// TIA Portal V15.1 export
// export: Created 2024-06-21T08:41:19.7465003Z, ExportSetting WithDefaults, DisplayName Totally Integrated Automation Portal, DisplayVersion V15.1 Update 5, DisplayName TIA Portal Openness, DisplayVersion V15.1 Update 5, DisplayName SINAMICS Startdrive Advanced, DisplayVersion V15.1, DisplayName G130, G150, S120, S150, SINAMICS MV, S210, DisplayVersion V15.1, DisplayName G110M, G120, G120C, G120D, G120P, DisplayVersion V15.1, DisplayName STEP 7 Professional, DisplayVersion V15.1 Update 5, DisplayName STEP 7 Safety, DisplayVersion V15.1, DisplayName WinCC Professional, DisplayVersion V15.1 Update 5, DisplayName SIMATIC Visualization Architect, DisplayVersion V15.1
FUNCTION_BLOCK "LGBTurnTable2W2S-MoviFitFCPN"   // FB6698, FBD
TITLE = LGBMovUnit2Pos2W2S-MoviFitFCPN / LGBTurnTable2W2S-MoviFitFCPN
{ S7_Optimized_Access := 'TRUE' }
AUTHOR : VCC
FAMILY : Tooling
VERSION : 0.1
// ============================================================================
// This module will be used for a unit with 2 stop positions, 2 speeds and controlled by a 
// SEW MOVIFIT-FC fieldbus frequency converter.
// It will get commands from higher level, evaluate the status of the interlock 
// and give a finished in return when the task is completed.
// It will get commands from higher level, evaluate the status of the interlock 
// and give a finished in return when the task is completed.
// ===========================================================================
// stored: AutoNumber false, IsIECCheckEnabled false, IsRetainMemResEnabled false, MemoryReserve 100, SetENOAutomatically False, UDAEnableTagReadback false
   VAR_INPUT
      I_PosSet { ExternalAccessible := 'False'; ExternalVisible := 'False'; ExternalWritable := 'False'} : Bool;   // Position Set Detection
      I_LowSpeedSet { ExternalAccessible := 'False'; ExternalVisible := 'False'; ExternalWritable := 'False'} : Bool;   // Low Speed Detection Set
      I_PosRes { ExternalAccessible := 'False'; ExternalVisible := 'False'; ExternalWritable := 'False'} : Bool;   // Position Reset Detection
      I_LowSpeedRes { ExternalAccessible := 'False'; ExternalVisible := 'False'; ExternalWritable := 'False'} : Bool;   // Low Speed Detection Reset
      I_SetBegin { ExternalAccessible := 'False'; ExternalVisible := 'False'; ExternalWritable := 'False'} : Bool;   // Function Set begin selection
      I_ResBegin { ExternalAccessible := 'False'; ExternalVisible := 'False'; ExternalWritable := 'False'} : Bool;   // Function Reset begin selection
      I_PBSet { ExternalAccessible := 'False'; ExternalVisible := 'False'; ExternalWritable := 'False'} : Bool;   // Push button for Set direction used in manual
      I_PBReset { ExternalAccessible := 'False'; ExternalVisible := 'False'; ExternalWritable := 'False'} : Bool;   // Push button for reset direcion used in manual
      I_SetIntlkOK { ExternalAccessible := 'False'; ExternalVisible := 'False'; ExternalWritable := 'False'} : Bool;   // Set Interlock
      I_ResIntlkOK { ExternalAccessible := 'False'; ExternalVisible := 'False'; ExternalWritable := 'False'} : Bool;   // Reset Interlock
      I_MotorProtection { ExternalAccessible := 'False'; ExternalVisible := 'False'; ExternalWritable := 'False'} : Bool;   // Motor protection
      I_ReleaseBrake { ExternalAccessible := 'False'; ExternalVisible := 'False'; ExternalWritable := 'False'} : Bool;   // Release brake
      I_SafetyOk { ExternalAccessible := 'False'; ExternalVisible := 'False'; ExternalWritable := 'False'} : Bool;   // Safety Ok
      I_MotionStopOk { ExternalAccessible := 'False'; ExternalVisible := 'False'; ExternalWritable := 'False'} : Bool;   // Safety Ok / The motion stop is Ok
      I_LowSpeed { ExternalAccessible := 'False'; ExternalVisible := 'False'; ExternalWritable := 'False'} : Real;   // Low speed Value (set-up %)
      I_HighSpeed { ExternalAccessible := 'False'; ExternalVisible := 'False'; ExternalWritable := 'False'} : Real;   // High speed Value (set-up %)
      I_SafetyStatusWord { ExternalAccessible := 'False'; ExternalVisible := 'False'; ExternalWritable := 'False'} : Word;   // Safety Status
      I_SafetyControlWord { ExternalAccessible := 'False'; ExternalVisible := 'False'; ExternalWritable := 'False'} : Word;   // Safety Control Word
   END_VAR
   VAR_OUTPUT
      O_SumPosSet { ExternalAccessible := 'False'; ExternalVisible := 'False'; ExternalWritable := 'False'} : Bool;   // Summary In Position Set
      O_SumPosRes { ExternalAccessible := 'False'; ExternalVisible := 'False'; ExternalWritable := 'False'} : Bool;   // Summary In Position Reset
      O_ReleaseBrake { ExternalAccessible := 'False'; ExternalVisible := 'False'; ExternalWritable := 'False'} : Bool;   // Release the brake of the motor
      O_Active { ExternalAccessible := 'False'; ExternalVisible := 'False'; ExternalWritable := 'False'} : Bool;   // Motor Active
      O_FuncRunning { ExternalAccessible := 'False'; ExternalVisible := 'False'; ExternalWritable := 'False'} : Bool;   // Signal that the function is busy
      O_SetFinished { ExternalAccessible := 'False'; ExternalVisible := 'False'; ExternalWritable := 'False'} : Bool;   // Function Set finished to Master Sequencing
      O_ResFinished { ExternalAccessible := 'False'; ExternalVisible := 'False'; ExternalWritable := 'False'} : Bool;   // Function Reset finished to Master Sequencing
      O_LEDSet { ExternalAccessible := 'False'; ExternalVisible := 'False'; ExternalWritable := 'False'} : Bool;   // Ledindication / Led indication for Set
      O_LEDRes { ExternalAccessible := 'False'; ExternalVisible := 'False'; ExternalWritable := 'False'} : Bool;   // Ledindication / Led indication for Reset
      O_ReadyForOperation { ExternalAccessible := 'False'; ExternalVisible := 'False'; ExternalWritable := 'False'} : Bool;   // Ready for operation
      O_AlarmABCondition { ExternalAccessible := 'False'; ExternalVisible := 'False'; ExternalWritable := 'False'} : Bool;   // Alarm AB Condition
      O_AlarmA { ExternalAccessible := 'False'; ExternalVisible := 'False'; ExternalWritable := 'False'} : Bool;   // Alarm A
      O_AlarmB { ExternalAccessible := 'False'; ExternalVisible := 'False'; ExternalWritable := 'False'} : Bool;   // Alarm B
      O_AlarmC { ExternalAccessible := 'False'; ExternalVisible := 'False'; ExternalWritable := 'False'} : Bool;   // Alarm C
      O_AlarmD { ExternalAccessible := 'False'; ExternalVisible := 'False'; ExternalWritable := 'False'} : Bool;   // Alarm D
      H_AlarmDWord { ExternalAccessible := 'False'; ExternalVisible := 'False'; ExternalWritable := 'False'} : DWord;   // Alarm Word
   END_VAR
   VAR_IN_OUT
      IO_Modes : "Modes";   // Modes
      H_HMI : "H_HMI";   // Animation
      "H_GBMovUnit2Pos2W2S-MoviFitFCPN" : "H_GBTurnTable2W2S-MoviFitFCPN";   // Animation
      C_Config : "TurnTable2W2S-MoviFitFCPNConfig";   // Config
   END_VAR
   VAR
      _MovFunc2Pos2s { ExternalAccessible := 'False'; ExternalVisible := 'False'; ExternalWritable := 'False'} : "LMovFnc2Pos2S";   // FB
      _StopPos { ExternalAccessible := 'False'; ExternalVisible := 'False'; ExternalWritable := 'False'} : "L2StopPos";   // FB
      _Motor { ExternalAccessible := 'False'; ExternalVisible := 'False'; ExternalWritable := 'False'} : "LGBMotor2W2S-MoviFitFCPN";   // FB
      H_FncSelInHMI { ExternalAccessible := 'False'; ExternalVisible := 'False'; ExternalWritable := 'False'} : Bool;
      AA_MotorProtection { ExternalAccessible := 'False'; ExternalVisible := 'False'; ExternalWritable := 'False'} : Bool;   // Motorprotection Not Ok
      AA_SafetySwitch { ExternalAccessible := 'False'; ExternalVisible := 'False'; ExternalWritable := 'False'} : Bool;   // Safety Switch Not Ok
      AB_STO { ExternalAccessible := 'False'; ExternalVisible := 'False'; ExternalWritable := 'False'} : Bool;   // Safety Switch Not Ok / Safety output to drive is active but no response from drive that the safety is ok
      AB_Alarm { ExternalAccessible := 'False'; ExternalVisible := 'False'; ExternalWritable := 'False'} : Bool;   // Frequency Control / Alarm Frequency Control
      AB_LSpeedDetSetMissing { ExternalAccessible := 'False'; ExternalVisible := 'False'; ExternalWritable := 'False'} : Bool;   // Low Speed Detector Set / Low Speed Detection Set Is Missing
      AB_LSpeedDetResMissing { ExternalAccessible := 'False'; ExternalVisible := 'False'; ExternalWritable := 'False'} : Bool;   // Low Speed Detector Reset / Low Speed Detection Reset Is Missing
      AB_KeepPosSetAlm { ExternalAccessible := 'False'; ExternalVisible := 'False'; ExternalWritable := 'False'} : Bool;   // Position Supervision Set Position / Lost Set Position
      AB_KeepPosResAlm { ExternalAccessible := 'False'; ExternalVisible := 'False'; ExternalWritable := 'False'} : Bool;   // Position Supervision Reset Position / Lost Reset Position
      AB_OvtSetAlm { ExternalAccessible := 'False'; ExternalVisible := 'False'; ExternalWritable := 'False'} : Bool;   // Timeout Set / TimeOut Set Direction
      AB_OvtResAlm { ExternalAccessible := 'False'; ExternalVisible := 'False'; ExternalWritable := 'False'} : Bool;   // Timeout Reset / TimeOut Reset Direction
      AB_TwoDetAlm { ExternalAccessible := 'False'; ExternalVisible := 'False'; ExternalWritable := 'False'} : Bool;   // Set Reset Activated Simultaneously / Detection Set & Reset Activated Simultaneously
      AC_KeepPosSetAlm { ExternalAccessible := 'False'; ExternalVisible := 'False'; ExternalWritable := 'False'} : Bool;   // Lost Set Position
      AC_KeepPosResAlm { ExternalAccessible := 'False'; ExternalVisible := 'False'; ExternalWritable := 'False'} : Bool;   // Lost Reset Position
      AC_OvtSetAlm { ExternalAccessible := 'False'; ExternalVisible := 'False'; ExternalWritable := 'False'} : Bool;   // Timeout Set / TimeOut Set Direction
      AC_OvtResAlm { ExternalAccessible := 'False'; ExternalVisible := 'False'; ExternalWritable := 'False'} : Bool;   // Timeout Reset / TimeOut Reset Direction
      AC_TwoDetAlm { ExternalAccessible := 'False'; ExternalVisible := 'False'; ExternalWritable := 'False'} : Bool;   // Set Reset Activated Simultaneously / Detection Set & Reset Activated Simultaneously
      AD_OvtSetWarn { ExternalAccessible := 'False'; ExternalVisible := 'False'; ExternalWritable := 'False'} : Bool;   // Timeout Set / TimeOut Set Direction
      AD_OvtResWarn { ExternalAccessible := 'False'; ExternalVisible := 'False'; ExternalWritable := 'False'} : Bool;   // Timeout Reset / TimeOut Reset Direction
      AD_IntlkSetAlm { ExternalAccessible := 'False'; ExternalVisible := 'False'; ExternalWritable := 'False'} : Bool;   // Interlock Set
      AD_IntlkResAlm { ExternalAccessible := 'False'; ExternalVisible := 'False'; ExternalWritable := 'False'} : Bool;   // Interlock Reset
      AD_Warning { ExternalAccessible := 'False'; ExternalVisible := 'False'; ExternalWritable := 'False'} : Bool;   // Frequency Control / Warning Frequency Control
      AA_NoBusControl { ExternalAccessible := 'False'; ExternalVisible := 'False'; ExternalWritable := 'False'} : Bool;   // Bus control inactive / Bus Control Inactive Frequency Control
      AD_MotionStop { ExternalAccessible := 'False'; ExternalVisible := 'False'; ExternalWritable := 'False'} : Bool;   // Motion Stop
      AC_ConfigCalibrationAlm { ExternalAccessible := 'False'; ExternalVisible := 'False'; ExternalWritable := 'False'} : Bool;   // The Config values for Warming/Alarm time must be ALL zero or ALL different from zero
      AD_CalibrationWarn { ExternalAccessible := 'False'; ExternalVisible := 'False'; ExternalWritable := 'False'} : Bool;   // No High speed selected so Calibration is not possible
      AC_ConfigRampAlm { ExternalAccessible := 'False'; ExternalVisible := 'False'; ExternalWritable := 'False'} : Bool;   // The config value for the ramp is not correct, must be zero or the config values for the calculation of the ramp must be ALL zero
      AC_ConfigRampCalcAlm { ExternalAccessible := 'False'; ExternalVisible := 'False'; ExternalWritable := 'False'} : Bool;   // The config values for the calculation of the ramp must be ALL different from zero
      PODataNotEnabled { ExternalAccessible := 'False'; ExternalVisible := 'False'; ExternalWritable := 'False'} : Bool;   // Bus control inactive
      SafetyOk { ExternalAccessible := 'False'; ExternalVisible := 'False'; ExternalWritable := 'False'} : Bool;   // Safety Ok
      AlarmABCondition { ExternalAccessible := 'False'; ExternalVisible := 'False'; ExternalWritable := 'False'} : Bool;   // Alarm AB Condition
   END_VAR
   VAR RETAIN
      LowSpeedDetSetOk { ExternalAccessible := 'False'; ExternalVisible := 'False'; ExternalWritable := 'False'} : Bool;   // Low speed Set detector ok
      LowSpeedDetResOk { ExternalAccessible := 'False'; ExternalVisible := 'False'; ExternalWritable := 'False'} : Bool;   // Low speed Reset detector ok
   END_VAR
   VAR
      SetPos { ExternalAccessible := 'False'; ExternalVisible := 'False'; ExternalWritable := 'False'} : Bool;   // Set position
      ResPos { ExternalAccessible := 'False'; ExternalVisible := 'False'; ExternalWritable := 'False'} : Bool;   // Reset position
      AlarmA { ExternalAccessible := 'False'; ExternalVisible := 'False'; ExternalWritable := 'False'} : Bool;   // Alarm A
      AlarmB { ExternalAccessible := 'False'; ExternalVisible := 'False'; ExternalWritable := 'False'} : Bool;   // Alarm B
      AlarmC { ExternalAccessible := 'False'; ExternalVisible := 'False'; ExternalWritable := 'False'} : Bool;   // Alarm C
      AlarmD { ExternalAccessible := 'False'; ExternalVisible := 'False'; ExternalWritable := 'False'} : Bool;   // Alarm D
      FuncRunning { ExternalAccessible := 'False'; ExternalVisible := 'False'; ExternalWritable := 'False'} : Bool;   // Function running
      MovFuncAlmCond { ExternalAccessible := 'False'; ExternalVisible := 'False'; ExternalWritable := 'False'} : Bool;   // Move function Alarm Condition
      StopPosAlmCond { ExternalAccessible := 'False'; ExternalVisible := 'False'; ExternalWritable := 'False'} : Bool;   // Stop posistion Alarm Condition
      KeepPosSetAlm { ExternalAccessible := 'False'; ExternalVisible := 'False'; ExternalWritable := 'False'} : Bool;   // Alarm Keep Position Set Position
      KeepPosResAlm { ExternalAccessible := 'False'; ExternalVisible := 'False'; ExternalWritable := 'False'} : Bool;   // Position Supervision Reset Position
      OvtSetAlm { ExternalAccessible := 'False'; ExternalVisible := 'False'; ExternalWritable := 'False'} : Bool;   // Timeout Set
      OvtResAlm { ExternalAccessible := 'False'; ExternalVisible := 'False'; ExternalWritable := 'False'} : Bool;   // Overtime reset Alarm
      TwoDetAlm { ExternalAccessible := 'False'; ExternalVisible := 'False'; ExternalWritable := 'False'} : Bool;   // Set Reset Activated Simultaneously
      OutOfUse { ExternalAccessible := 'False'; ExternalVisible := 'False'; ExternalWritable := 'False'} : Bool;   // Out of use
      MotorLoopAlarmCond { ExternalAccessible := 'False'; ExternalVisible := 'False'; ExternalWritable := 'False'} : Bool;   // Motor loop Alarm Condition
      SafetySwNc { ExternalAccessible := 'False'; ExternalVisible := 'False'; ExternalWritable := 'False'} : Bool;   // Safety switch NC
      InitDirection { ExternalAccessible := 'False'; ExternalVisible := 'False'; ExternalWritable := 'False'} : Bool;   // Init Direction
      ReadyForOperation { ExternalAccessible := 'False'; ExternalVisible := 'False'; ExternalWritable := 'False'} : Bool;   // Motor Loop Ready for operation
      MotorLoopActive { ExternalAccessible := 'False'; ExternalVisible := 'False'; ExternalWritable := 'False'} : Bool;   // Motor Loop Active
      ReleaseBrake { ExternalAccessible := 'False'; ExternalVisible := 'False'; ExternalWritable := 'False'} : Bool;   // Release brake
      CmdSet { ExternalAccessible := 'False'; ExternalVisible := 'False'; ExternalWritable := 'False'} : Bool;   // Command set
      CmdRes { ExternalAccessible := 'False'; ExternalVisible := 'False'; ExternalWritable := 'False'} : Bool;   // DCommand Reset
      MotorCmdHSpdSet { ExternalAccessible := 'False'; ExternalVisible := 'False'; ExternalWritable := 'False'} : Bool;   // Command high speed to motorloop set
      MotorCmdLSpdSet { ExternalAccessible := 'False'; ExternalVisible := 'False'; ExternalWritable := 'False'} : Bool;   // Command low speed to motorloop set
      MotorCmdHSpdRes { ExternalAccessible := 'False'; ExternalVisible := 'False'; ExternalWritable := 'False'} : Bool;   // Command high speed to motorloop reset
      MotorCmdLSpdRes { ExternalAccessible := 'False'; ExternalVisible := 'False'; ExternalWritable := 'False'} : Bool;   // Command low speed to motorloop reset
      DetStopHSpdSetMem { ExternalAccessible := 'False'; ExternalVisible := 'False'; ExternalWritable := 'False'} : Bool;   // Memorisation stop high speed set
      DetStopHSpdResMem { ExternalAccessible := 'False'; ExternalVisible := 'False'; ExternalWritable := 'False'} : Bool;   // Memorisation stop high speed reset
      ManLowSpdSel { ExternalAccessible := 'False'; ExternalVisible := 'False'; ExternalWritable := 'False'} : Bool;   // Low speed Selected in manual
      LowSpeedSetDetMissingCond { ExternalAccessible := 'False'; ExternalVisible := 'False'; ExternalWritable := 'False'} : Bool;   // Low speed detector missing condition set
      LowSpeedResDetMissingCond { ExternalAccessible := 'False'; ExternalVisible := 'False'; ExternalWritable := 'False'} : Bool;   // Low speed detector missing condition reset
      SetIntlkOK { ExternalAccessible := 'False'; ExternalVisible := 'False'; ExternalWritable := 'False'} : Bool;   // Set Interlock
      ResIntlkOK { ExternalAccessible := 'False'; ExternalVisible := 'False'; ExternalWritable := 'False'} : Bool;   // Reset Interlock
      Edge { ExternalAccessible := 'False'; ExternalVisible := 'False'; ExternalWritable := 'False'} : Array[1..8] of Bool;
   END_VAR
   VAR_TEMP
      H_HMITemp : "H_HMI";   // Animation
      HMICMD : "ConvHMICMD";
      H_HMIMotor : "H_HMI";
      TempDInt : DInt;   // Temp DInt
   END_VAR
   VAR_TEMP   // added for the SCL form of the ladder/FBD networks
      _w1 : Bool;
   END_VAR
BEGIN

REGION Network 1: **** 1 - Inputs **** HMI Commands
   // HMI Commands
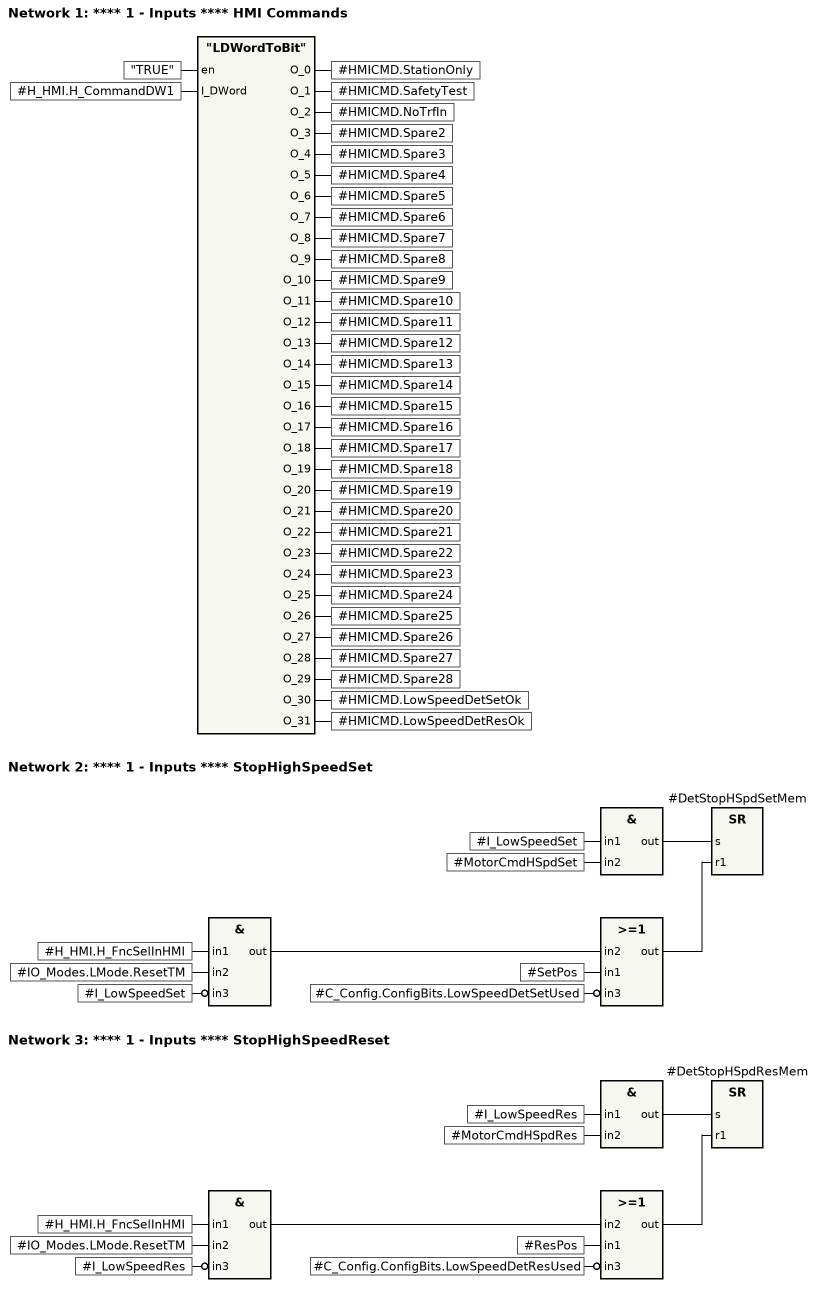
   IF "TRUE" THEN
       "LDWordToBit"(I_DWord := #H_HMI.H_CommandDW1,
                     O_0 => #HMICMD.StationOnly,
                     O_1 => #HMICMD.SafetyTest,
                     O_2 => #HMICMD.NoTrfIn,
                     O_3 => #HMICMD.Spare2,
                     O_4 => #HMICMD.Spare3,
                     O_5 => #HMICMD.Spare4,
                     O_6 => #HMICMD.Spare5,
                     O_7 => #HMICMD.Spare6,
                     O_8 => #HMICMD.Spare7,
                     O_9 => #HMICMD.Spare8,
                     O_10 => #HMICMD.Spare9,
                     O_11 => #HMICMD.Spare10,
                     O_12 => #HMICMD.Spare11,
                     O_13 => #HMICMD.Spare12,
                     O_14 => #HMICMD.Spare13,
                     O_15 => #HMICMD.Spare14,
                     O_16 => #HMICMD.Spare15,
                     O_17 => #HMICMD.Spare16,
                     O_18 => #HMICMD.Spare17,
                     O_19 => #HMICMD.Spare18,
                     O_20 => #HMICMD.Spare19,
                     O_21 => #HMICMD.Spare20,
                     O_22 => #HMICMD.Spare21,
                     O_23 => #HMICMD.Spare22,
                     O_24 => #HMICMD.Spare23,
                     O_25 => #HMICMD.Spare24,
                     O_26 => #HMICMD.Spare25,
                     O_27 => #HMICMD.Spare26,
                     O_28 => #HMICMD.Spare27,
                     O_29 => #HMICMD.Spare28,
                     O_30 => #HMICMD.LowSpeedDetSetOk,
                     O_31 => #HMICMD.LowSpeedDetResOk);
   END_IF;
END_REGION

REGION Network 2: **** 1 - Inputs **** StopHighSpeedSet
   // Stop high speed set memorisation (go to low speed)
   IF #I_LowSpeedSet AND #MotorCmdHSpdSet THEN
       #DetStopHSpdSetMem := TRUE;   // SR flip-flop
   END_IF;
   IF (#H_HMI.H_FncSelInHMI AND #IO_Modes.LMode.ResetTM AND NOT #I_LowSpeedSet) OR #SetPos OR NOT #C_Config.ConfigBits.LowSpeedDetSetUsed THEN
       #DetStopHSpdSetMem := FALSE;
   END_IF;
END_REGION

REGION Network 3: **** 1 - Inputs **** StopHighSpeedReset
   // Stop high speed reset memorisation (go to low speed)
   IF #I_LowSpeedRes AND #MotorCmdHSpdRes THEN
       #DetStopHSpdResMem := TRUE;   // SR flip-flop
   END_IF;
   IF (#H_HMI.H_FncSelInHMI AND #IO_Modes.LMode.ResetTM AND NOT #I_LowSpeedRes) OR #ResPos OR NOT #C_Config.ConfigBits.LowSpeedDetResUsed THEN
       #DetStopHSpdResMem := FALSE;
   END_IF;
END_REGION

REGION Network 4: **** 1 - Inputs **** LowSpeedSet
   // Low speed set detector been on
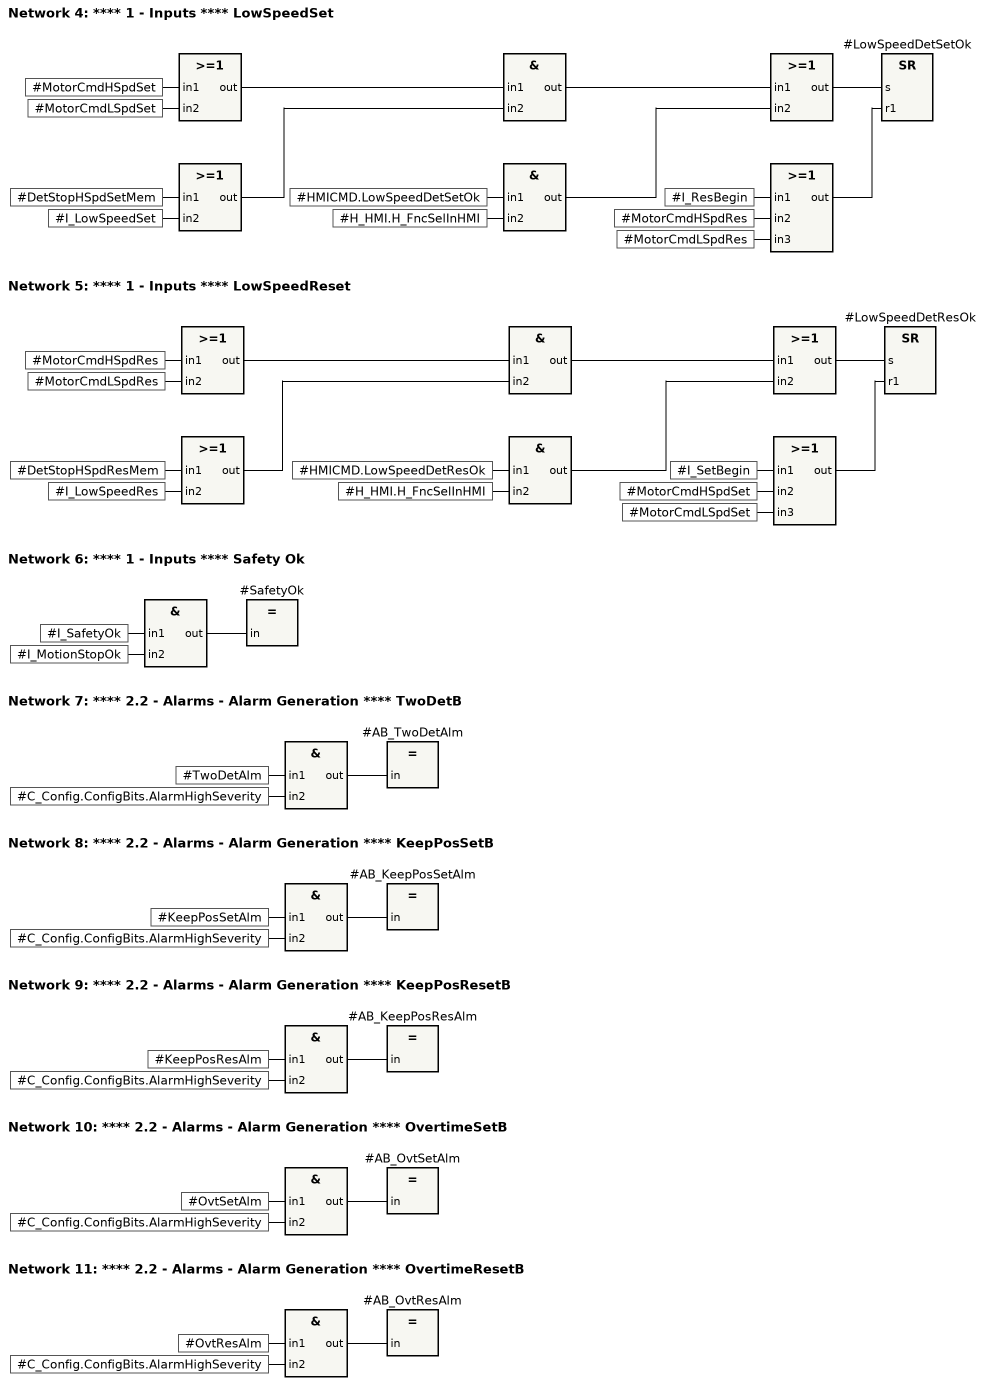
   IF ((#MotorCmdHSpdSet OR #MotorCmdLSpdSet) AND (#DetStopHSpdSetMem OR #I_LowSpeedSet)) OR (#HMICMD.LowSpeedDetSetOk AND #H_HMI.H_FncSelInHMI) THEN
       #LowSpeedDetSetOk := TRUE;   // SR flip-flop
   END_IF;
   IF #I_ResBegin OR #MotorCmdHSpdRes OR #MotorCmdLSpdRes THEN #LowSpeedDetSetOk := FALSE; END_IF;
END_REGION

REGION Network 5: **** 1 - Inputs **** LowSpeedReset
   // Low speed reset detector been on
   IF ((#MotorCmdHSpdRes OR #MotorCmdLSpdRes) AND (#DetStopHSpdResMem OR #I_LowSpeedRes)) OR (#HMICMD.LowSpeedDetResOk AND #H_HMI.H_FncSelInHMI) THEN
       #LowSpeedDetResOk := TRUE;   // SR flip-flop
   END_IF;
   IF #I_SetBegin OR #MotorCmdHSpdSet OR #MotorCmdLSpdSet THEN #LowSpeedDetResOk := FALSE; END_IF;
END_REGION

REGION Network 6: **** 1 - Inputs **** Safety Ok
   #SafetyOk := #I_SafetyOk AND #I_MotionStopOk;
END_REGION

REGION Network 7: **** 2.2 - Alarms - Alarm Generation **** TwoDetB
   // Two Detection B Alarm
   #AB_TwoDetAlm := #TwoDetAlm AND #C_Config.ConfigBits.AlarmHighSeverity;
END_REGION

REGION Network 8: **** 2.2 - Alarms - Alarm Generation **** KeepPosSetB
   // Keep position Set B Alarm
   #AB_KeepPosSetAlm := #KeepPosSetAlm AND #C_Config.ConfigBits.AlarmHighSeverity;
END_REGION

REGION Network 9: **** 2.2 - Alarms - Alarm Generation **** KeepPosResetB
   // Keep position reset B Alarm
   #AB_KeepPosResAlm := #KeepPosResAlm AND #C_Config.ConfigBits.AlarmHighSeverity;
END_REGION

REGION Network 10: **** 2.2 - Alarms - Alarm Generation **** OvertimeSetB
   // Overtime set B Alarm
   #AB_OvtSetAlm := #OvtSetAlm AND #C_Config.ConfigBits.AlarmHighSeverity;
END_REGION

REGION Network 11: **** 2.2 - Alarms - Alarm Generation **** OvertimeResetB
   // Overtime reset B Alarm
   #AB_OvtResAlm := #OvtResAlm AND #C_Config.ConfigBits.AlarmHighSeverity;
END_REGION

REGION Network 12: **** 2.2 - Alarms - Alarm Generation **** TwoDetC
   // Two Detection C Alarm
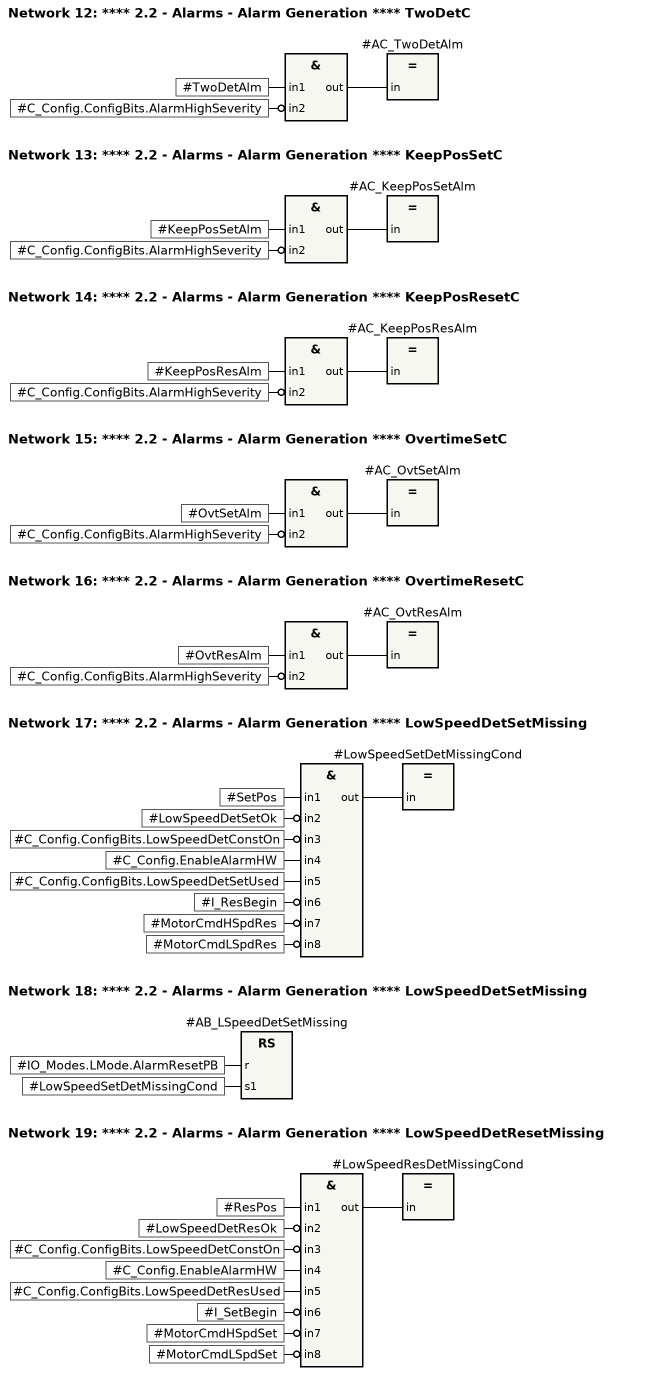
   #AC_TwoDetAlm := #TwoDetAlm AND NOT #C_Config.ConfigBits.AlarmHighSeverity;
END_REGION

REGION Network 13: **** 2.2 - Alarms - Alarm Generation **** KeepPosSetC
   // Keep position Set C Alarm
   #AC_KeepPosSetAlm := #KeepPosSetAlm AND NOT #C_Config.ConfigBits.AlarmHighSeverity;
END_REGION

REGION Network 14: **** 2.2 - Alarms - Alarm Generation **** KeepPosResetC
   // Keep position reset C Alarm
   #AC_KeepPosResAlm := #KeepPosResAlm AND NOT #C_Config.ConfigBits.AlarmHighSeverity;
END_REGION

REGION Network 15: **** 2.2 - Alarms - Alarm Generation **** OvertimeSetC
   // Overtime set C Alarm
   #AC_OvtSetAlm := #OvtSetAlm AND NOT #C_Config.ConfigBits.AlarmHighSeverity;
END_REGION

REGION Network 16: **** 2.2 - Alarms - Alarm Generation **** OvertimeResetC
   // Overtime reset C Alarm
   #AC_OvtResAlm := #OvtResAlm AND NOT #C_Config.ConfigBits.AlarmHighSeverity;
END_REGION

REGION Network 17: **** 2.2 - Alarms - Alarm Generation **** LowSpeedDetSetMissing
   // Alarm LowSpeed detector set missing
   #LowSpeedSetDetMissingCond := #SetPos AND NOT #LowSpeedDetSetOk AND NOT #C_Config.ConfigBits.LowSpeedDetConstOn AND #C_Config.EnableAlarmHW AND #C_Config.ConfigBits.LowSpeedDetSetUsed AND NOT #I_ResBegin AND NOT #MotorCmdHSpdRes AND NOT #MotorCmdLSpdRes;
END_REGION

REGION Network 18: **** 2.2 - Alarms - Alarm Generation **** LowSpeedDetSetMissing
   // Alarm LowSpeed detector set missing
   IF #IO_Modes.LMode.AlarmResetPB THEN
       #AB_LSpeedDetSetMissing := FALSE;   // RS flip-flop
   END_IF;
   IF #LowSpeedSetDetMissingCond THEN #AB_LSpeedDetSetMissing := TRUE; END_IF;
END_REGION

REGION Network 19: **** 2.2 - Alarms - Alarm Generation **** LowSpeedDetResetMissing
   // Alarm LowSpeed detector reset missing
   #LowSpeedResDetMissingCond := #ResPos AND NOT #LowSpeedDetResOk AND NOT #C_Config.ConfigBits.LowSpeedDetConstOn AND #C_Config.EnableAlarmHW AND #C_Config.ConfigBits.LowSpeedDetResUsed AND NOT #I_SetBegin AND NOT #MotorCmdHSpdSet AND NOT #MotorCmdLSpdSet;
END_REGION

REGION Network 20: **** 2.2 - Alarms - Alarm Generation **** LowSpeedDetResetMissing
   // Alarm LowSpeed detector reset missing
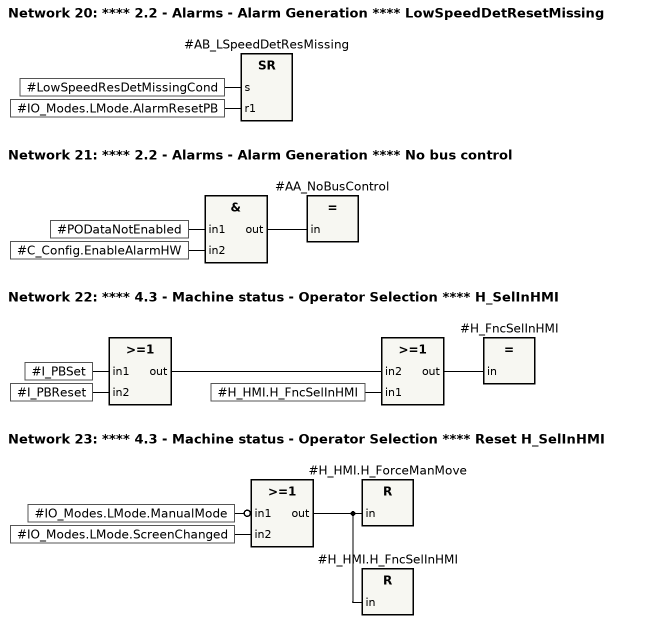
   IF #LowSpeedResDetMissingCond THEN
       #AB_LSpeedDetResMissing := TRUE;   // SR flip-flop
   END_IF;
   IF #IO_Modes.LMode.AlarmResetPB THEN #AB_LSpeedDetResMissing := FALSE; END_IF;
END_REGION

REGION Network 21: **** 2.2 - Alarms - Alarm Generation **** No bus control
   #AA_NoBusControl := #PODataNotEnabled AND #C_Config.EnableAlarmHW;
END_REGION

REGION Network 22: **** 4.3 - Machine status - Operator Selection **** H_SelInHMI
   #H_FncSelInHMI := #I_PBSet OR #I_PBReset OR #H_HMI.H_FncSelInHMI;
END_REGION

REGION Network 23: **** 4.3 - Machine status - Operator Selection **** Reset H_SelInHMI
   // Reset H_SelInHMI
   IF NOT #IO_Modes.LMode.ManualMode OR #IO_Modes.LMode.ScreenChanged THEN
       #H_HMI.H_ForceManMove := FALSE;
       #H_HMI.H_FncSelInHMI := FALSE;
   END_IF;
END_REGION

REGION Network 24: **** 4.6 - Machine Status - Indication **** SetDetIAnim
   // Icon animation
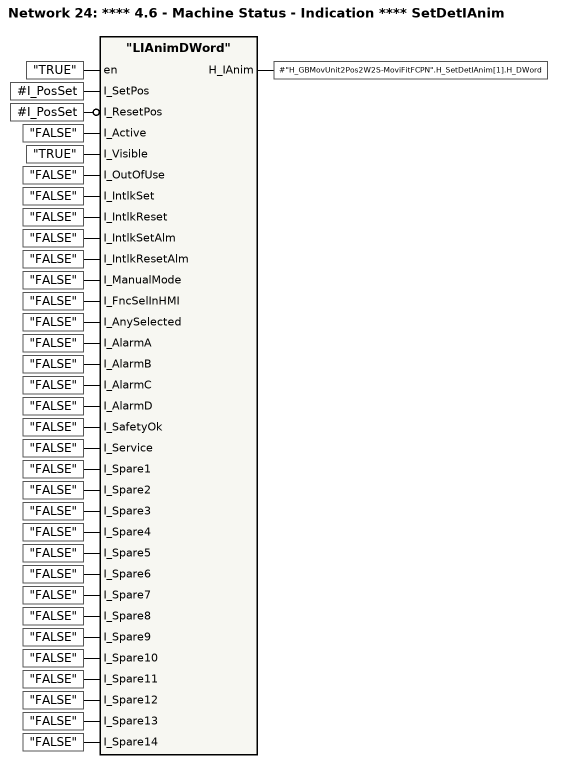
   IF "TRUE" THEN
       "LIAnimDWord"(I_SetPos := #I_PosSet,
                     I_ResetPos := NOT #I_PosSet,
                     I_Active := "FALSE",
                     I_Visible := "TRUE",
                     I_OutOfUse := "FALSE",
                     I_IntlkSet := "FALSE",
                     I_IntlkReset := "FALSE",
                     I_IntlkSetAlm := "FALSE",
                     I_IntlkResetAlm := "FALSE",
                     I_ManualMode := "FALSE",
                     I_FncSelInHMI := "FALSE",
                     I_AnySelected := "FALSE",
                     I_AlarmA := "FALSE",
                     I_AlarmB := "FALSE",
                     I_AlarmC := "FALSE",
                     I_AlarmD := "FALSE",
                     I_SafetyOk := "FALSE",
                     I_Service := "FALSE",
                     I_Spare1 := "FALSE",
                     I_Spare2 := "FALSE",
                     I_Spare3 := "FALSE",
                     I_Spare4 := "FALSE",
                     I_Spare5 := "FALSE",
                     I_Spare6 := "FALSE",
                     I_Spare7 := "FALSE",
                     I_Spare8 := "FALSE",
                     I_Spare9 := "FALSE",
                     I_Spare10 := "FALSE",
                     I_Spare11 := "FALSE",
                     I_Spare12 := "FALSE",
                     I_Spare13 := "FALSE",
                     I_Spare14 := "FALSE",
                     H_IAnim => #"H_GBMovUnit2Pos2W2S-MoviFitFCPN".H_SetDetIAnim[1].H_DWord);
   END_IF;
END_REGION

REGION Network 25: **** 4.6 - Machine Status - Indication **** ResetDetIAnim
   // Icon animation
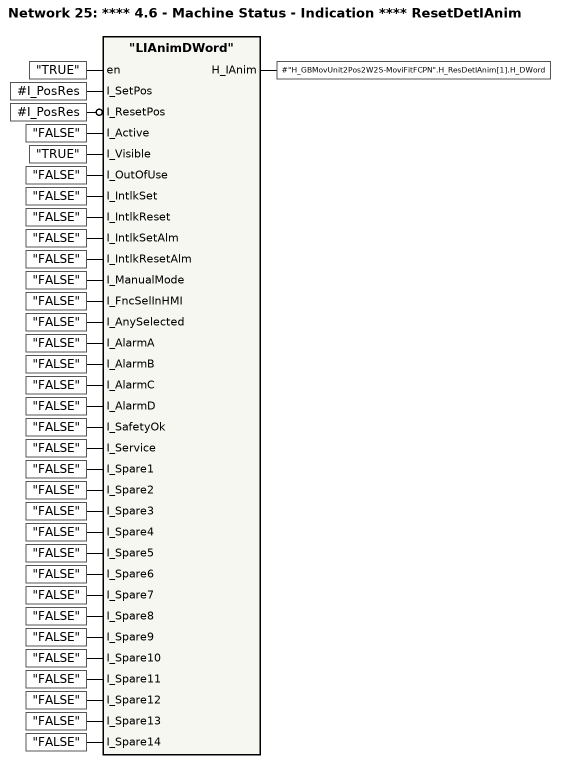
   IF "TRUE" THEN
       "LIAnimDWord"(I_SetPos := #I_PosRes,
                     I_ResetPos := NOT #I_PosRes,
                     I_Active := "FALSE",
                     I_Visible := "TRUE",
                     I_OutOfUse := "FALSE",
                     I_IntlkSet := "FALSE",
                     I_IntlkReset := "FALSE",
                     I_IntlkSetAlm := "FALSE",
                     I_IntlkResetAlm := "FALSE",
                     I_ManualMode := "FALSE",
                     I_FncSelInHMI := "FALSE",
                     I_AnySelected := "FALSE",
                     I_AlarmA := "FALSE",
                     I_AlarmB := "FALSE",
                     I_AlarmC := "FALSE",
                     I_AlarmD := "FALSE",
                     I_SafetyOk := "FALSE",
                     I_Service := "FALSE",
                     I_Spare1 := "FALSE",
                     I_Spare2 := "FALSE",
                     I_Spare3 := "FALSE",
                     I_Spare4 := "FALSE",
                     I_Spare5 := "FALSE",
                     I_Spare6 := "FALSE",
                     I_Spare7 := "FALSE",
                     I_Spare8 := "FALSE",
                     I_Spare9 := "FALSE",
                     I_Spare10 := "FALSE",
                     I_Spare11 := "FALSE",
                     I_Spare12 := "FALSE",
                     I_Spare13 := "FALSE",
                     I_Spare14 := "FALSE",
                     H_IAnim => #"H_GBMovUnit2Pos2W2S-MoviFitFCPN".H_ResDetIAnim[1].H_DWord);
   END_IF;
END_REGION

REGION Network 26: **** 4.6 - Machine Status - Indication **** LSpdDetSetIAnim
   // Icon animation
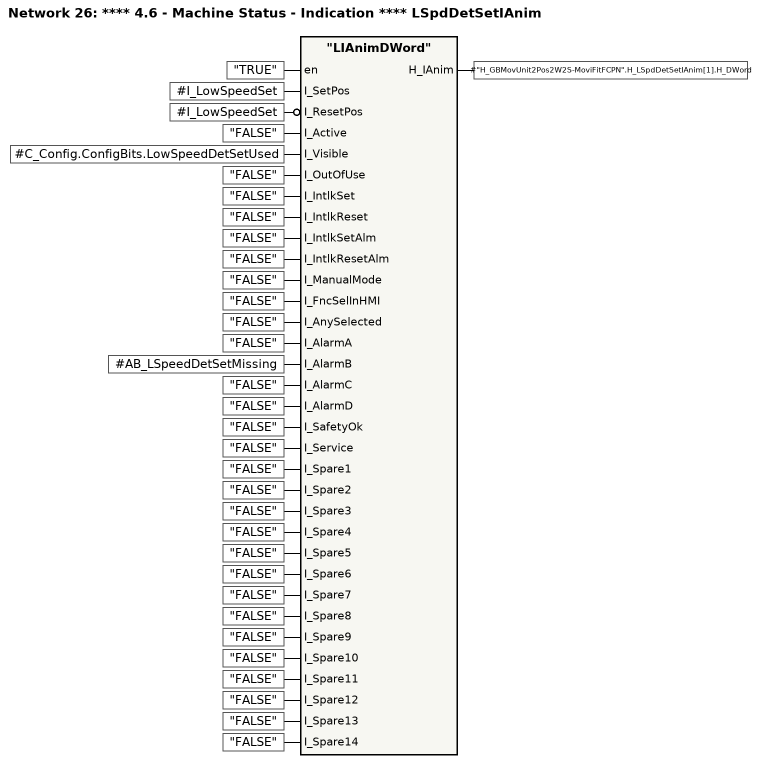
   IF "TRUE" THEN
       "LIAnimDWord"(I_SetPos := #I_LowSpeedSet,
                     I_ResetPos := NOT #I_LowSpeedSet,
                     I_Active := "FALSE",
                     I_Visible := #C_Config.ConfigBits.LowSpeedDetSetUsed,
                     I_OutOfUse := "FALSE",
                     I_IntlkSet := "FALSE",
                     I_IntlkReset := "FALSE",
                     I_IntlkSetAlm := "FALSE",
                     I_IntlkResetAlm := "FALSE",
                     I_ManualMode := "FALSE",
                     I_FncSelInHMI := "FALSE",
                     I_AnySelected := "FALSE",
                     I_AlarmA := "FALSE",
                     I_AlarmB := #AB_LSpeedDetSetMissing,
                     I_AlarmC := "FALSE",
                     I_AlarmD := "FALSE",
                     I_SafetyOk := "FALSE",
                     I_Service := "FALSE",
                     I_Spare1 := "FALSE",
                     I_Spare2 := "FALSE",
                     I_Spare3 := "FALSE",
                     I_Spare4 := "FALSE",
                     I_Spare5 := "FALSE",
                     I_Spare6 := "FALSE",
                     I_Spare7 := "FALSE",
                     I_Spare8 := "FALSE",
                     I_Spare9 := "FALSE",
                     I_Spare10 := "FALSE",
                     I_Spare11 := "FALSE",
                     I_Spare12 := "FALSE",
                     I_Spare13 := "FALSE",
                     I_Spare14 := "FALSE",
                     H_IAnim => #"H_GBMovUnit2Pos2W2S-MoviFitFCPN".H_LSpdDetSetIAnim[1].H_DWord);
   END_IF;
END_REGION

REGION Network 27: **** 4.6 - Machine Status - Indication **** LSpdDetResIAnim
   // Icon animation
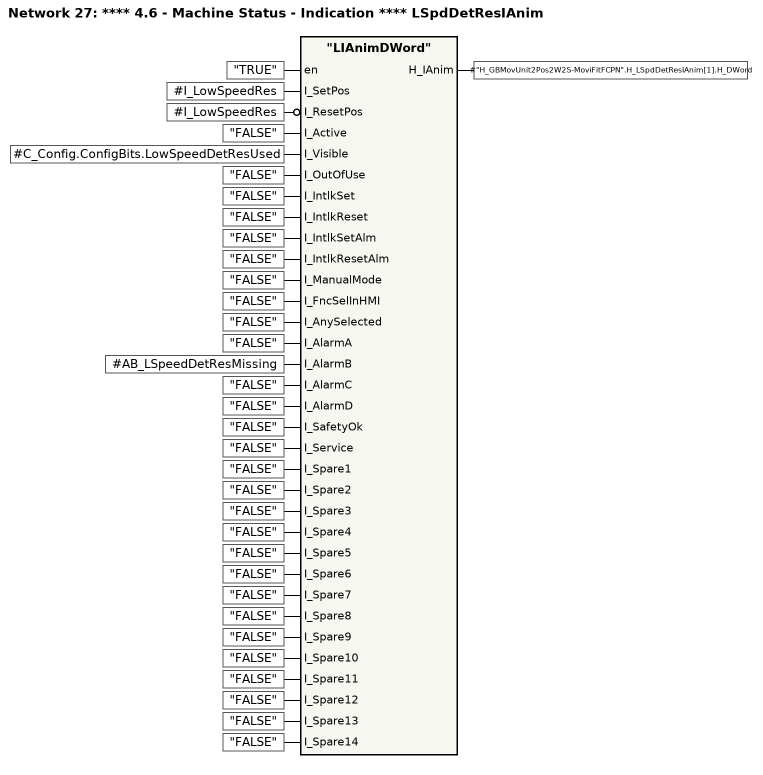
   IF "TRUE" THEN
       "LIAnimDWord"(I_SetPos := #I_LowSpeedRes,
                     I_ResetPos := NOT #I_LowSpeedRes,
                     I_Active := "FALSE",
                     I_Visible := #C_Config.ConfigBits.LowSpeedDetResUsed,
                     I_OutOfUse := "FALSE",
                     I_IntlkSet := "FALSE",
                     I_IntlkReset := "FALSE",
                     I_IntlkSetAlm := "FALSE",
                     I_IntlkResetAlm := "FALSE",
                     I_ManualMode := "FALSE",
                     I_FncSelInHMI := "FALSE",
                     I_AnySelected := "FALSE",
                     I_AlarmA := "FALSE",
                     I_AlarmB := #AB_LSpeedDetResMissing,
                     I_AlarmC := "FALSE",
                     I_AlarmD := "FALSE",
                     I_SafetyOk := "FALSE",
                     I_Service := "FALSE",
                     I_Spare1 := "FALSE",
                     I_Spare2 := "FALSE",
                     I_Spare3 := "FALSE",
                     I_Spare4 := "FALSE",
                     I_Spare5 := "FALSE",
                     I_Spare6 := "FALSE",
                     I_Spare7 := "FALSE",
                     I_Spare8 := "FALSE",
                     I_Spare9 := "FALSE",
                     I_Spare10 := "FALSE",
                     I_Spare11 := "FALSE",
                     I_Spare12 := "FALSE",
                     I_Spare13 := "FALSE",
                     I_Spare14 := "FALSE",
                     H_IAnim => #"H_GBMovUnit2Pos2W2S-MoviFitFCPN".H_LSpdDetResIAnim[1].H_DWord);
   END_IF;
END_REGION

REGION Network 28: **** 4.6 - Machine Status - Indication **** Icon Animation
   // Icon animation
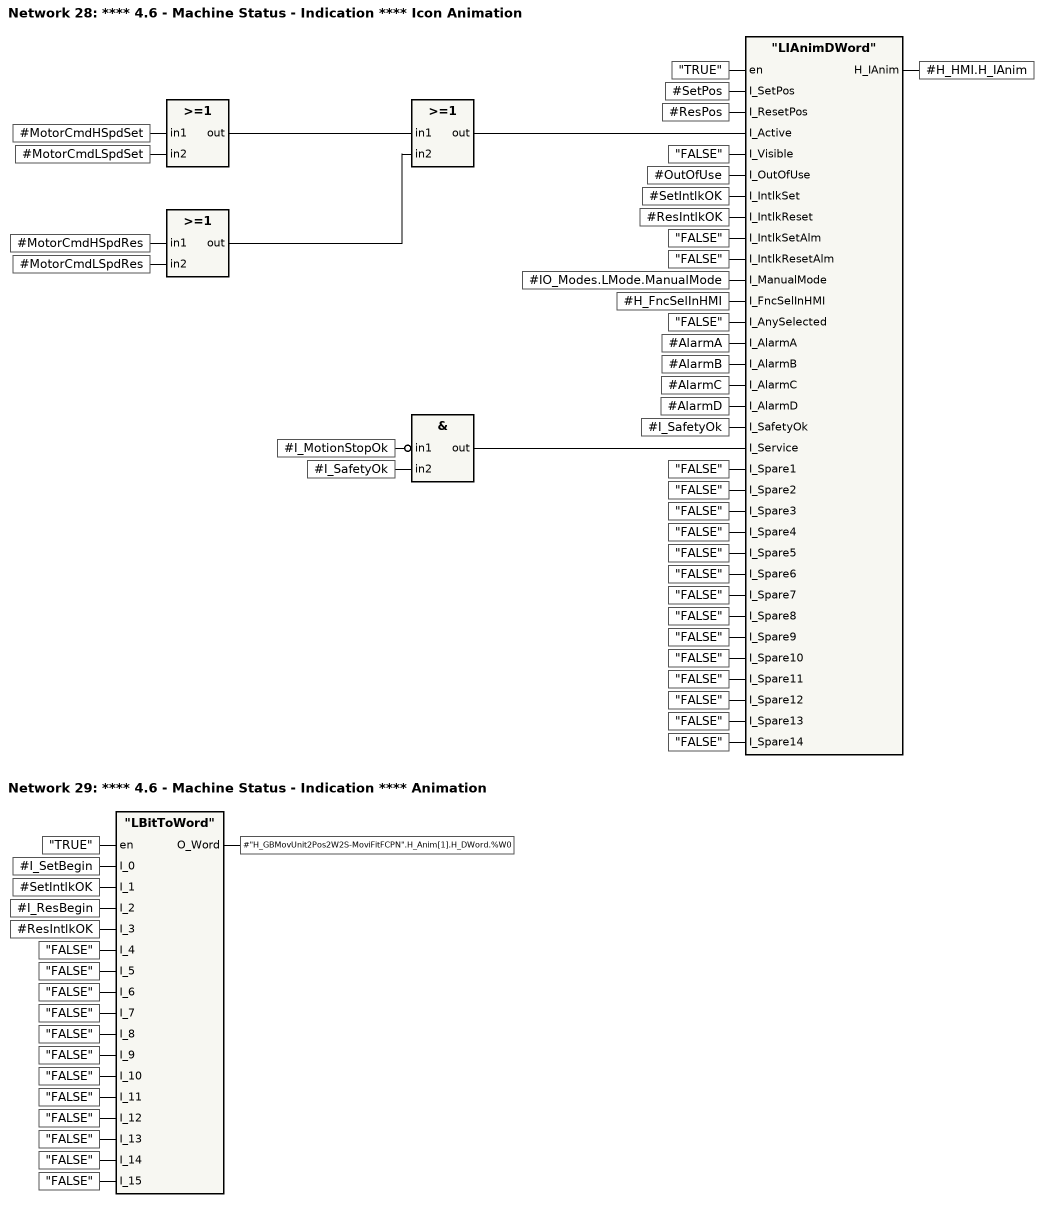
   IF "TRUE" THEN
       "LIAnimDWord"(I_SetPos := #SetPos,
                     I_ResetPos := #ResPos,
                     I_Active := #MotorCmdHSpdSet OR #MotorCmdLSpdSet OR #MotorCmdHSpdRes OR #MotorCmdLSpdRes,
                     I_Visible := "FALSE",
                     I_OutOfUse := #OutOfUse,
                     I_IntlkSet := #SetIntlkOK,
                     I_IntlkReset := #ResIntlkOK,
                     I_IntlkSetAlm := "FALSE",
                     I_IntlkResetAlm := "FALSE",
                     I_ManualMode := #IO_Modes.LMode.ManualMode,
                     I_FncSelInHMI := #H_FncSelInHMI,
                     I_AnySelected := "FALSE",
                     I_AlarmA := #AlarmA,
                     I_AlarmB := #AlarmB,
                     I_AlarmC := #AlarmC,
                     I_AlarmD := #AlarmD,
                     I_SafetyOk := #I_SafetyOk,
                     I_Service := NOT #I_MotionStopOk AND #I_SafetyOk,
                     I_Spare1 := "FALSE",
                     I_Spare2 := "FALSE",
                     I_Spare3 := "FALSE",
                     I_Spare4 := "FALSE",
                     I_Spare5 := "FALSE",
                     I_Spare6 := "FALSE",
                     I_Spare7 := "FALSE",
                     I_Spare8 := "FALSE",
                     I_Spare9 := "FALSE",
                     I_Spare10 := "FALSE",
                     I_Spare11 := "FALSE",
                     I_Spare12 := "FALSE",
                     I_Spare13 := "FALSE",
                     I_Spare14 := "FALSE",
                     H_IAnim => #H_HMI.H_IAnim);
   END_IF;
END_REGION

REGION Network 29: **** 4.6 - Machine Status - Indication **** Animation
   // Animation
   IF "TRUE" THEN
       "LBitToWord"(I_0 := #I_SetBegin,
                    I_1 := #SetIntlkOK,
                    I_2 := #I_ResBegin,
                    I_3 := #ResIntlkOK,
                    I_4 := "FALSE",
                    I_5 := "FALSE",
                    I_6 := "FALSE",
                    I_7 := "FALSE",
                    I_8 := "FALSE",
                    I_9 := "FALSE",
                    I_10 := "FALSE",
                    I_11 := "FALSE",
                    I_12 := "FALSE",
                    I_13 := "FALSE",
                    I_14 := "FALSE",
                    I_15 := "FALSE",
                    O_Word => #"H_GBMovUnit2Pos2W2S-MoviFitFCPN".H_Anim[1].H_DWord.%W0);
   END_IF;
END_REGION

REGION Network 30: **** 4.6 - Machine Status - Indication **** Animation
   // Animation
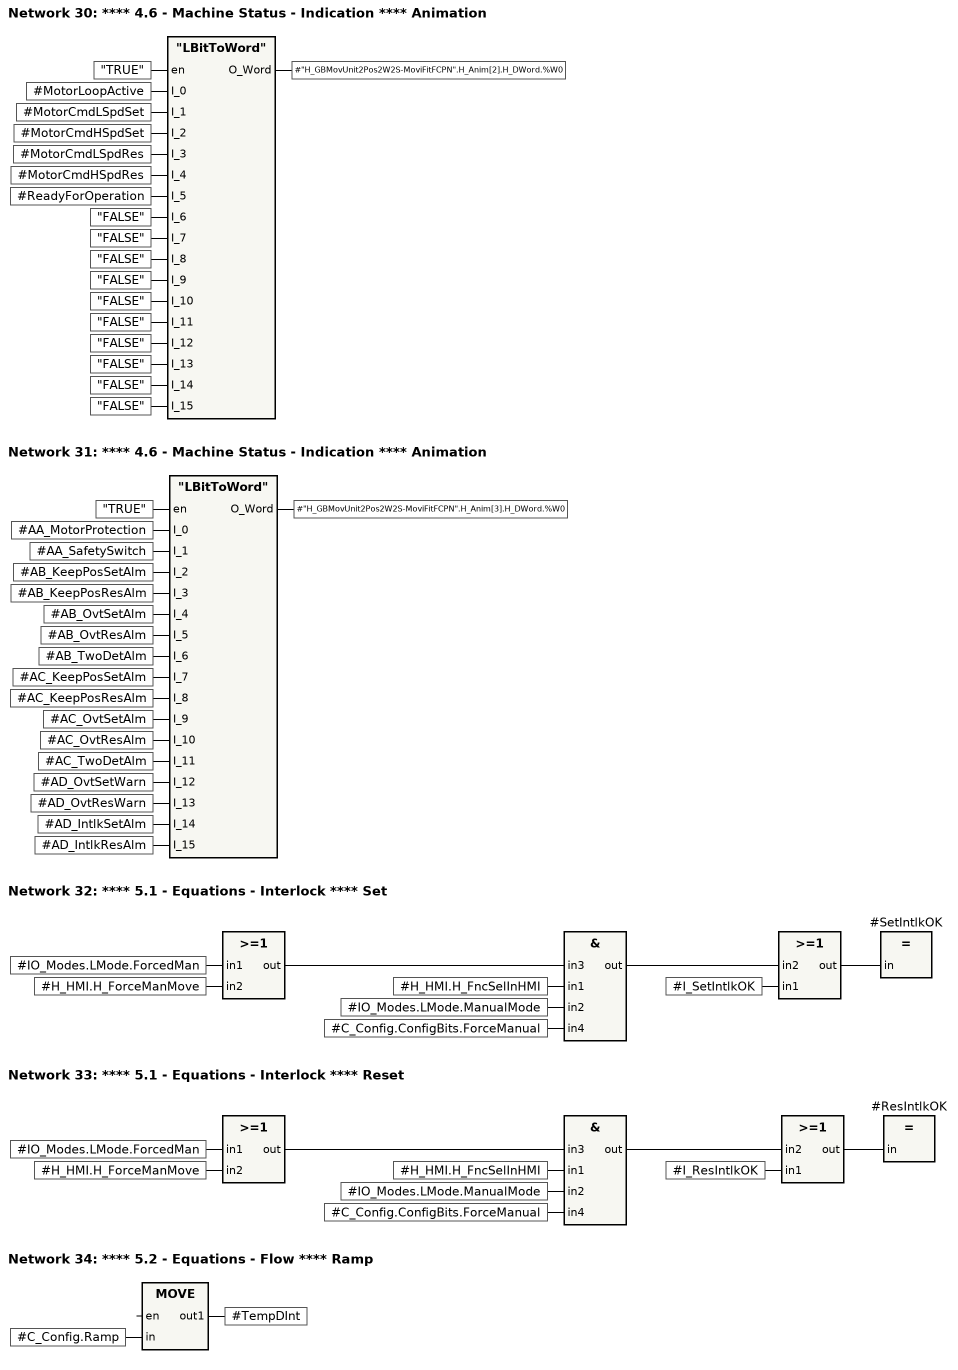
   IF "TRUE" THEN
       "LBitToWord"(I_0 := #MotorLoopActive,
                    I_1 := #MotorCmdLSpdSet,
                    I_2 := #MotorCmdHSpdSet,
                    I_3 := #MotorCmdLSpdRes,
                    I_4 := #MotorCmdHSpdRes,
                    I_5 := #ReadyForOperation,
                    I_6 := "FALSE",
                    I_7 := "FALSE",
                    I_8 := "FALSE",
                    I_9 := "FALSE",
                    I_10 := "FALSE",
                    I_11 := "FALSE",
                    I_12 := "FALSE",
                    I_13 := "FALSE",
                    I_14 := "FALSE",
                    I_15 := "FALSE",
                    O_Word => #"H_GBMovUnit2Pos2W2S-MoviFitFCPN".H_Anim[2].H_DWord.%W0);
   END_IF;
END_REGION

REGION Network 31: **** 4.6 - Machine Status - Indication **** Animation
   // Animation
   IF "TRUE" THEN
       "LBitToWord"(I_0 := #AA_MotorProtection,
                    I_1 := #AA_SafetySwitch,
                    I_2 := #AB_KeepPosSetAlm,
                    I_3 := #AB_KeepPosResAlm,
                    I_4 := #AB_OvtSetAlm,
                    I_5 := #AB_OvtResAlm,
                    I_6 := #AB_TwoDetAlm,
                    I_7 := #AC_KeepPosSetAlm,
                    I_8 := #AC_KeepPosResAlm,
                    I_9 := #AC_OvtSetAlm,
                    I_10 := #AC_OvtResAlm,
                    I_11 := #AC_TwoDetAlm,
                    I_12 := #AD_OvtSetWarn,
                    I_13 := #AD_OvtResWarn,
                    I_14 := #AD_IntlkSetAlm,
                    I_15 := #AD_IntlkResAlm,
                    O_Word => #"H_GBMovUnit2Pos2W2S-MoviFitFCPN".H_Anim[3].H_DWord.%W0);
   END_IF;
END_REGION

REGION Network 32: **** 5.1 - Equations - Interlock **** Set
   // Interlock
   #SetIntlkOK := ((#IO_Modes.LMode.ForcedMan OR #H_HMI.H_ForceManMove) AND #H_HMI.H_FncSelInHMI AND #IO_Modes.LMode.ManualMode AND #C_Config.ConfigBits.ForceManual) OR #I_SetIntlkOK;
END_REGION

REGION Network 33: **** 5.1 - Equations - Interlock **** Reset
   // Interlock
   #ResIntlkOK := ((#IO_Modes.LMode.ForcedMan OR #H_HMI.H_ForceManMove) AND #H_HMI.H_FncSelInHMI AND #IO_Modes.LMode.ManualMode AND #C_Config.ConfigBits.ForceManual) OR #I_ResIntlkOK;
END_REGION

REGION Network 34: **** 5.2 - Equations - Flow **** Ramp
   #TempDInt := #C_Config.Ramp;
END_REGION

REGION Network 35: **** 7.2 - Submodule - Command Summary **** LowSpeedMan
   // Cmd summary low speed in manual
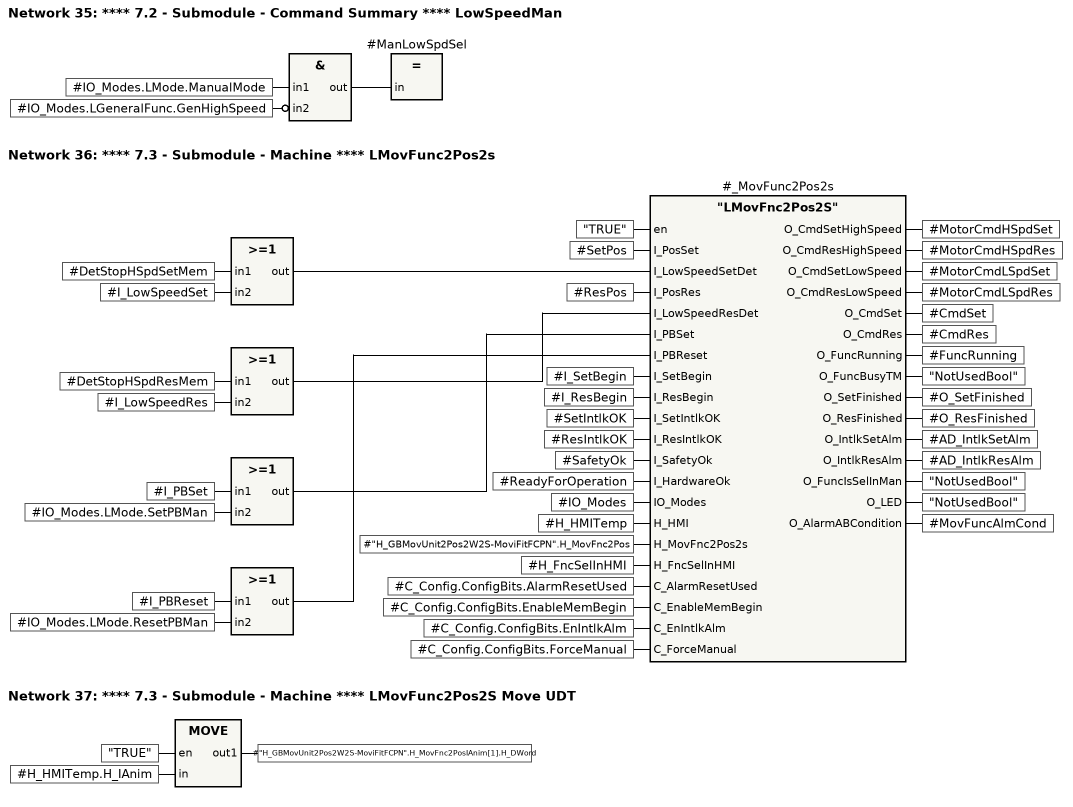
   #ManLowSpdSel := #IO_Modes.LMode.ManualMode AND NOT #IO_Modes.LGeneralFunc.GenHighSpeed;
END_REGION

REGION Network 36: **** 7.3 - Submodule - Machine **** LMovFunc2Pos2s
   // LMovFunc2Pos
   IF "TRUE" THEN
       #_MovFunc2Pos2s(I_PosSet := #SetPos,   // "LMovFnc2Pos2S"
                       I_LowSpeedSetDet := #DetStopHSpdSetMem OR #I_LowSpeedSet,
                       I_PosRes := #ResPos,
                       I_LowSpeedResDet := #DetStopHSpdResMem OR #I_LowSpeedRes,
                       I_PBSet := #I_PBSet OR #IO_Modes.LMode.SetPBMan,
                       I_PBReset := #I_PBReset OR #IO_Modes.LMode.ResetPBMan,
                       I_SetBegin := #I_SetBegin,
                       I_ResBegin := #I_ResBegin,
                       I_SetIntlkOK := #SetIntlkOK,
                       I_ResIntlkOK := #ResIntlkOK,
                       I_SafetyOk := #SafetyOk,
                       I_HardwareOk := #ReadyForOperation,
                       IO_Modes := #IO_Modes,
                       H_HMI := #H_HMITemp,
                       H_MovFnc2Pos2s := #"H_GBMovUnit2Pos2W2S-MoviFitFCPN".H_MovFnc2Pos,
                       H_FncSelInHMI := #H_FncSelInHMI,
                       C_AlarmResetUsed := #C_Config.ConfigBits.AlarmResetUsed,
                       C_EnableMemBegin := #C_Config.ConfigBits.EnableMemBegin,
                       C_EnIntlkAlm := #C_Config.ConfigBits.EnIntlkAlm,
                       C_ForceManual := #C_Config.ConfigBits.ForceManual,
                       O_CmdSetHighSpeed => #MotorCmdHSpdSet,
                       O_CmdResHighSpeed => #MotorCmdHSpdRes,
                       O_CmdSetLowSpeed => #MotorCmdLSpdSet,
                       O_CmdResLowSpeed => #MotorCmdLSpdRes,
                       O_CmdSet => #CmdSet,
                       O_CmdRes => #CmdRes,
                       O_FuncRunning => #FuncRunning,
                       O_FuncBusyTM => "NotUsedBool",
                       O_SetFinished => #O_SetFinished,
                       O_ResFinished => #O_ResFinished,
                       O_IntlkSetAlm => #AD_IntlkSetAlm,
                       O_IntlkResAlm => #AD_IntlkResAlm,
                       O_FuncIsSelInMan => "NotUsedBool",
                       O_LED => "NotUsedBool",
                       O_AlarmABCondition => #MovFuncAlmCond);
   END_IF;
END_REGION

REGION Network 37: **** 7.3 - Submodule - Machine **** LMovFunc2Pos2S Move UDT
   // LMovFunc2Pos2S Move UDT
   IF "TRUE" THEN
       #"H_GBMovUnit2Pos2W2S-MoviFitFCPN".H_MovFnc2PosIAnim[1].H_DWord := #H_HMITemp.H_IAnim;
   END_IF;
END_REGION

REGION Network 38: **** 7.3 - Submodule - Machine **** L2StopPos
   // L2StopPos
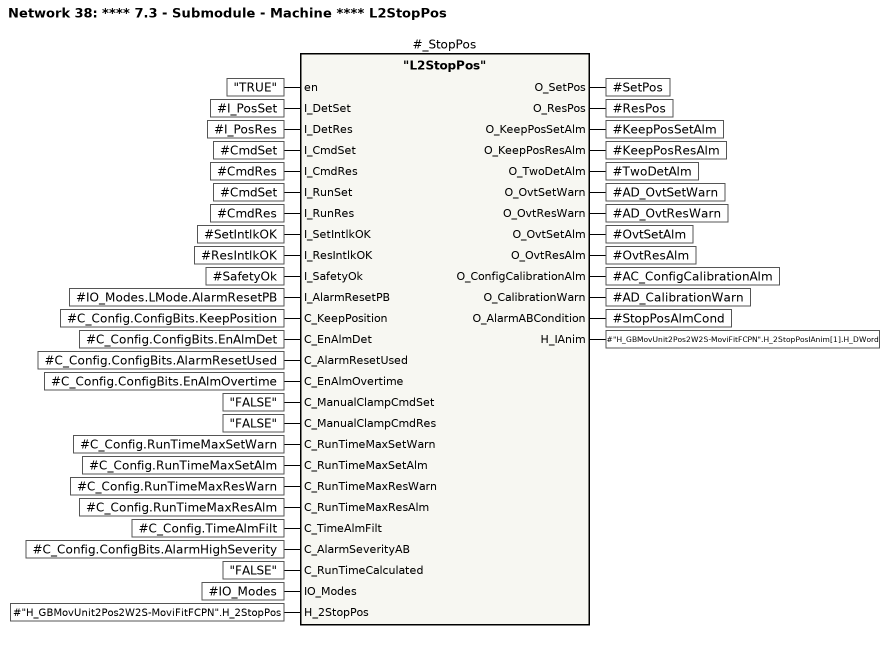
   IF "TRUE" THEN
       #_StopPos(I_DetSet := #I_PosSet,   // "L2StopPos"
                 I_DetRes := #I_PosRes,
                 I_CmdSet := #CmdSet,
                 I_CmdRes := #CmdRes,
                 I_RunSet := #CmdSet,
                 I_RunRes := #CmdRes,
                 I_SetIntlkOK := #SetIntlkOK,
                 I_ResIntlkOK := #ResIntlkOK,
                 I_SafetyOk := #SafetyOk,
                 I_AlarmResetPB := #IO_Modes.LMode.AlarmResetPB,
                 C_KeepPosition := #C_Config.ConfigBits.KeepPosition,
                 C_EnAlmDet := #C_Config.ConfigBits.EnAlmDet,
                 C_AlarmResetUsed := #C_Config.ConfigBits.AlarmResetUsed,
                 C_EnAlmOvertime := #C_Config.ConfigBits.EnAlmOvertime,
                 C_ManualClampCmdSet := "FALSE",
                 C_ManualClampCmdRes := "FALSE",
                 C_RunTimeMaxSetWarn := #C_Config.RunTimeMaxSetWarn,
                 C_RunTimeMaxSetAlm := #C_Config.RunTimeMaxSetAlm,
                 C_RunTimeMaxResWarn := #C_Config.RunTimeMaxResWarn,
                 C_RunTimeMaxResAlm := #C_Config.RunTimeMaxResAlm,
                 C_TimeAlmFilt := #C_Config.TimeAlmFilt,
                 C_AlarmSeverityAB := #C_Config.ConfigBits.AlarmHighSeverity,
                 C_RunTimeCalculated := "FALSE",
                 IO_Modes := #IO_Modes,
                 H_2StopPos := #"H_GBMovUnit2Pos2W2S-MoviFitFCPN".H_2StopPos,
                 O_SetPos => #SetPos,
                 O_ResPos => #ResPos,
                 O_KeepPosSetAlm => #KeepPosSetAlm,
                 O_KeepPosResAlm => #KeepPosResAlm,
                 O_TwoDetAlm => #TwoDetAlm,
                 O_OvtSetWarn => #AD_OvtSetWarn,
                 O_OvtResWarn => #AD_OvtResWarn,
                 O_OvtSetAlm => #OvtSetAlm,
                 O_OvtResAlm => #OvtResAlm,
                 O_ConfigCalibrationAlm => #AC_ConfigCalibrationAlm,
                 O_CalibrationWarn => #AD_CalibrationWarn,
                 O_AlarmABCondition => #StopPosAlmCond,
                 H_IAnim => #"H_GBMovUnit2Pos2W2S-MoviFitFCPN".H_2StopPosIAnim[1].H_DWord);
   END_IF;
END_REGION

REGION Network 39: **** 7.3 - Submodule - Machine **** Motor loop MOVIFIT-FC
   // Motor loop MOVIFIT-FC
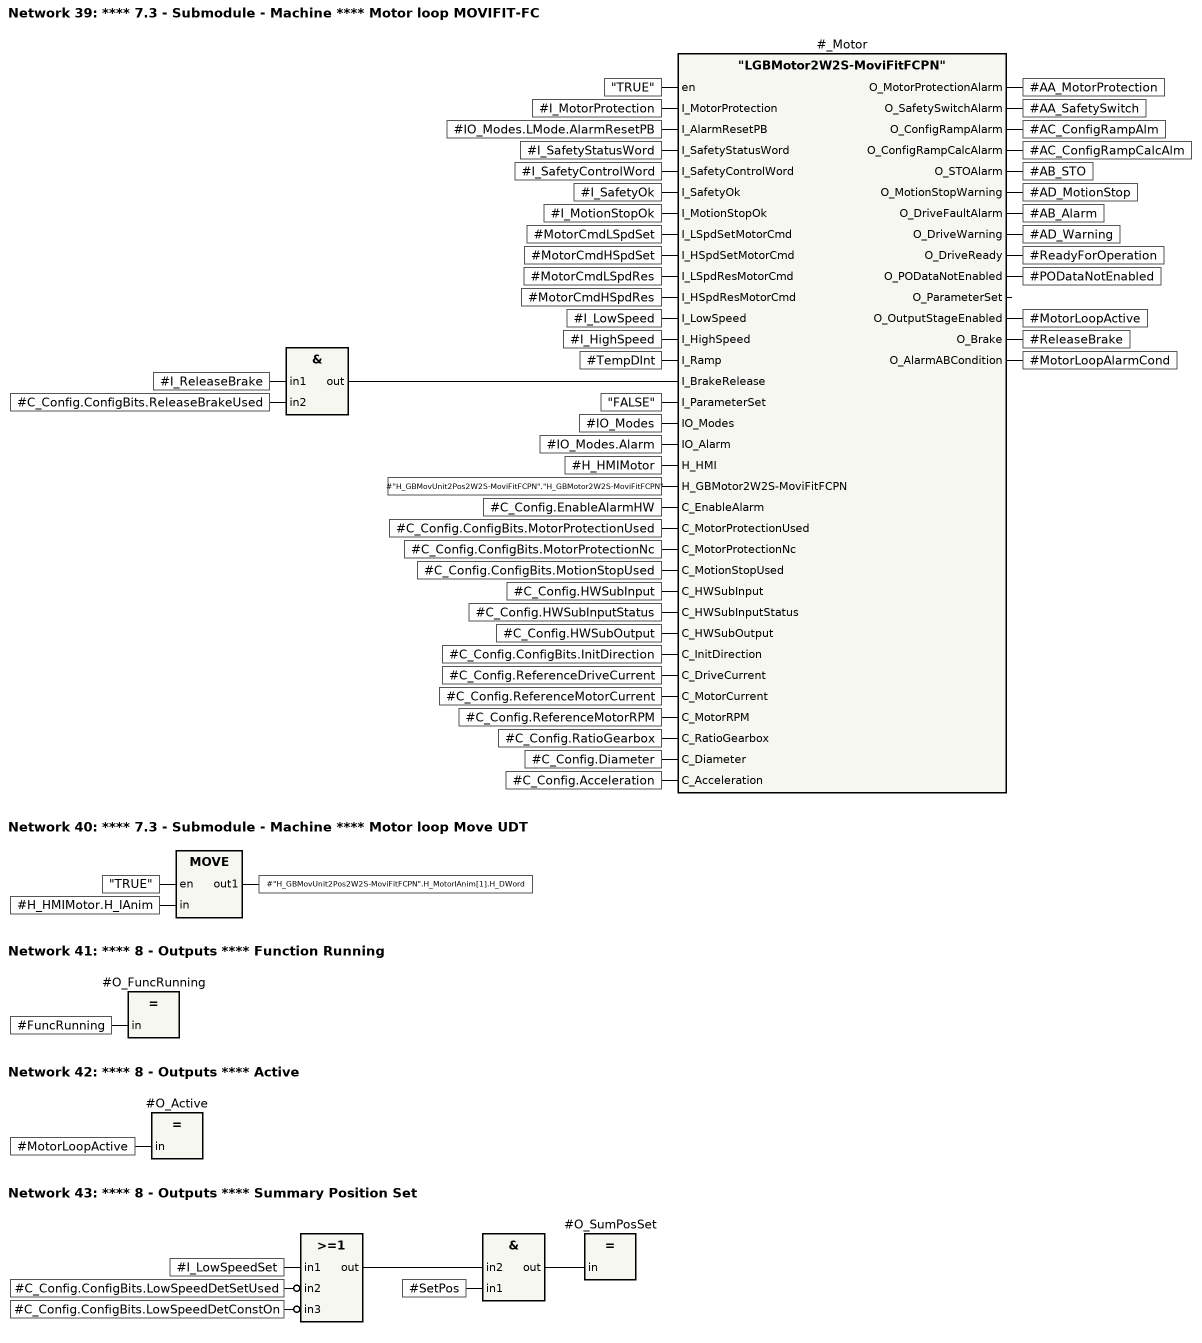
   IF "TRUE" THEN
       #_Motor(I_MotorProtection := #I_MotorProtection,   // "LGBMotor2W2S-MoviFitFCPN"
               I_AlarmResetPB := #IO_Modes.LMode.AlarmResetPB,
               I_SafetyStatusWord := #I_SafetyStatusWord,
               I_SafetyControlWord := #I_SafetyControlWord,
               I_SafetyOk := #I_SafetyOk,
               I_MotionStopOk := #I_MotionStopOk,
               I_LSpdSetMotorCmd := #MotorCmdLSpdSet,
               I_HSpdSetMotorCmd := #MotorCmdHSpdSet,
               I_LSpdResMotorCmd := #MotorCmdLSpdRes,
               I_HSpdResMotorCmd := #MotorCmdHSpdRes,
               I_LowSpeed := #I_LowSpeed,
               I_HighSpeed := #I_HighSpeed,
               I_Ramp := #TempDInt,
               I_BrakeRelease := #I_ReleaseBrake AND #C_Config.ConfigBits.ReleaseBrakeUsed,
               I_ParameterSet := "FALSE",
               IO_Modes := #IO_Modes,
               IO_Alarm := #IO_Modes.Alarm,
               H_HMI := #H_HMIMotor,
               "H_GBMotor2W2S-MoviFitFCPN" := #"H_GBMovUnit2Pos2W2S-MoviFitFCPN"."H_GBMotor2W2S-MoviFitFCPN",
               C_EnableAlarm := #C_Config.EnableAlarmHW,
               C_MotorProtectionUsed := #C_Config.ConfigBits.MotorProtectionUsed,
               C_MotorProtectionNc := #C_Config.ConfigBits.MotorProtectionNc,
               C_MotionStopUsed := #C_Config.ConfigBits.MotionStopUsed,
               C_HWSubInput := #C_Config.HWSubInput,
               C_HWSubInputStatus := #C_Config.HWSubInputStatus,
               C_HWSubOutput := #C_Config.HWSubOutput,
               C_InitDirection := #C_Config.ConfigBits.InitDirection,
               C_DriveCurrent := #C_Config.ReferenceDriveCurrent,
               C_MotorCurrent := #C_Config.ReferenceMotorCurrent,
               C_MotorRPM := #C_Config.ReferenceMotorRPM,
               C_RatioGearbox := #C_Config.RatioGearbox,
               C_Diameter := #C_Config.Diameter,
               C_Acceleration := #C_Config.Acceleration,
               O_MotorProtectionAlarm => #AA_MotorProtection,
               O_SafetySwitchAlarm => #AA_SafetySwitch,
               O_ConfigRampAlarm => #AC_ConfigRampAlm,
               O_ConfigRampCalcAlarm => #AC_ConfigRampCalcAlm,
               O_STOAlarm => #AB_STO,
               O_MotionStopWarning => #AD_MotionStop,
               O_DriveFaultAlarm => #AB_Alarm,
               O_DriveWarning => #AD_Warning,
               O_DriveReady => #ReadyForOperation,
               O_PODataNotEnabled => #PODataNotEnabled,
               O_OutputStageEnabled => #MotorLoopActive,
               O_Brake => #ReleaseBrake,
               O_AlarmABCondition => #MotorLoopAlarmCond);
   END_IF;
END_REGION

REGION Network 40: **** 7.3 - Submodule - Machine **** Motor loop Move UDT
   IF "TRUE" THEN #"H_GBMovUnit2Pos2W2S-MoviFitFCPN".H_MotorIAnim[1].H_DWord := #H_HMIMotor.H_IAnim; END_IF;
END_REGION

REGION Network 41: **** 8 - Outputs **** Function Running
   // Function Running
   #O_FuncRunning := #FuncRunning;
END_REGION

REGION Network 42: **** 8 - Outputs **** Active
   // Motor Loop active
   #O_Active := #MotorLoopActive;
END_REGION

REGION Network 43: **** 8 - Outputs **** Summary Position Set
   // Summary Position Set
   #O_SumPosSet := (#I_LowSpeedSet OR NOT #C_Config.ConfigBits.LowSpeedDetSetUsed OR NOT #C_Config.ConfigBits.LowSpeedDetConstOn) AND #SetPos;
END_REGION

REGION Network 44: **** 8 - Outputs **** Summary Position Set / **** 8 - Outputs **** Summary Position Reset
   // Summary Position Reset
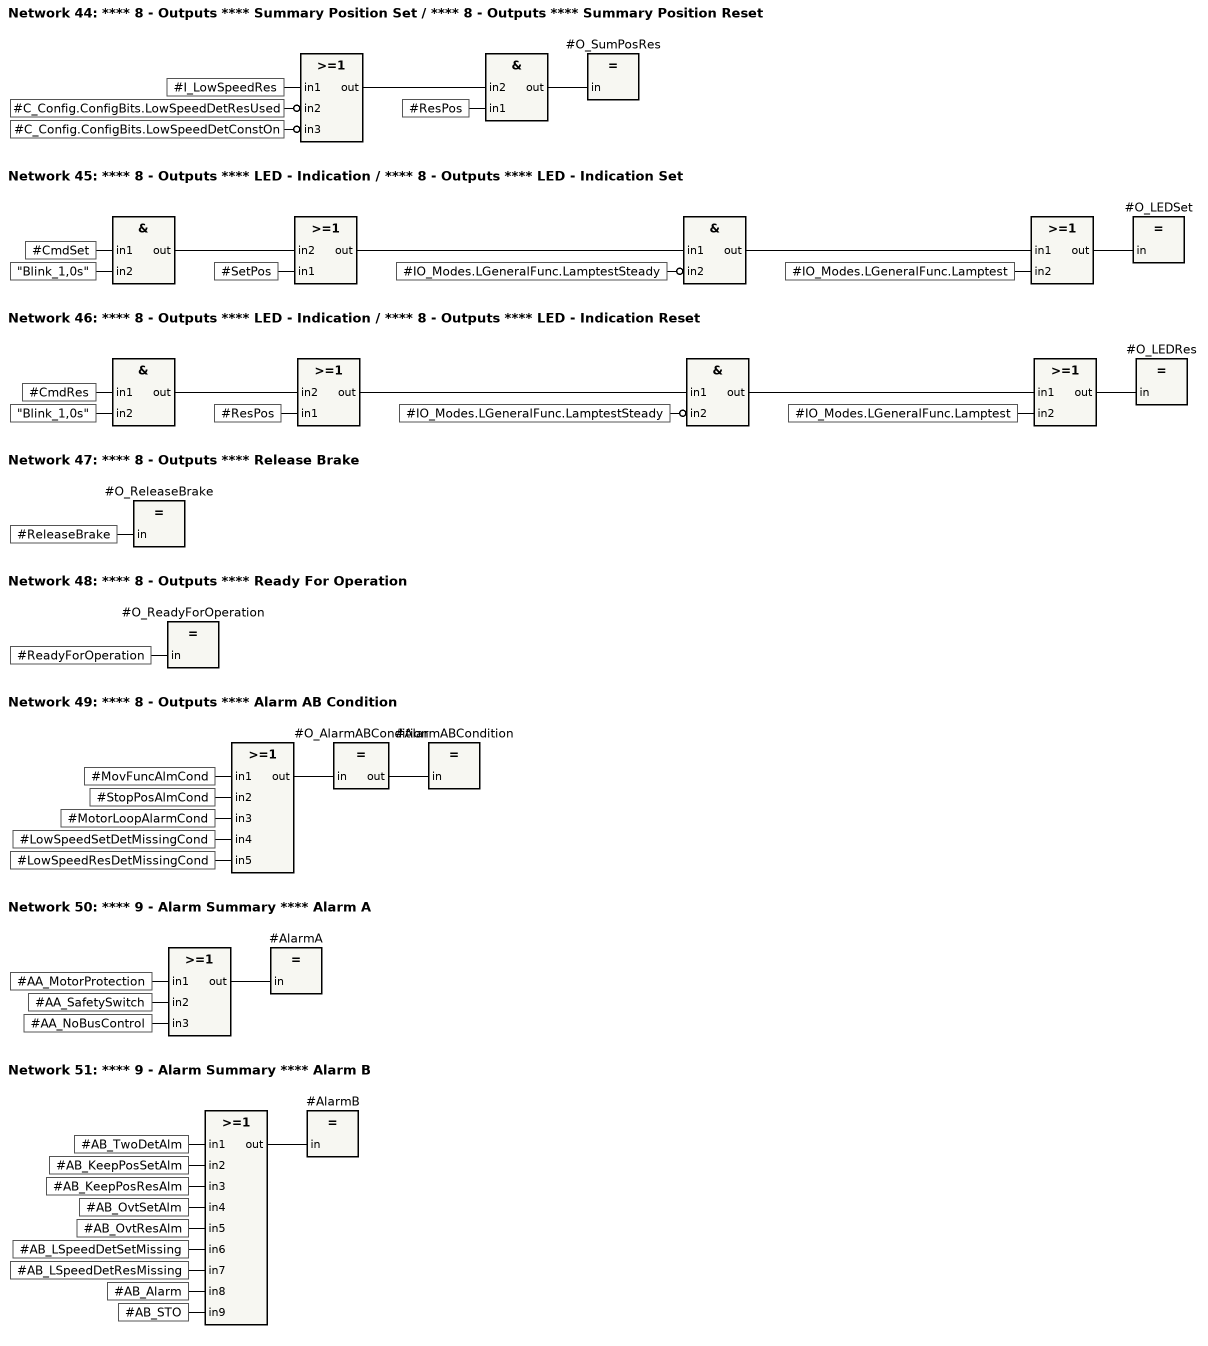
   #O_SumPosRes := (#I_LowSpeedRes OR NOT #C_Config.ConfigBits.LowSpeedDetResUsed OR NOT #C_Config.ConfigBits.LowSpeedDetConstOn) AND #ResPos;
END_REGION

REGION Network 45: **** 8 - Outputs **** LED - Indication / **** 8 - Outputs **** LED - Indication Set
   // LED - Indication
   #O_LEDSet := (((#CmdSet AND "Blink_1,0s") OR #SetPos) AND NOT #IO_Modes.LGeneralFunc.LamptestSteady) OR #IO_Modes.LGeneralFunc.Lamptest;
END_REGION

REGION Network 46: **** 8 - Outputs **** LED - Indication / **** 8 - Outputs **** LED - Indication Reset
   // LED - Indication
   #O_LEDRes := (((#CmdRes AND "Blink_1,0s") OR #ResPos) AND NOT #IO_Modes.LGeneralFunc.LamptestSteady) OR #IO_Modes.LGeneralFunc.Lamptest;
END_REGION

REGION Network 47: **** 8 - Outputs **** Release Brake
   // Release Brake
   #O_ReleaseBrake := #ReleaseBrake;
END_REGION

REGION Network 48: **** 8 - Outputs **** Ready For Operation
   // Ready For Operation
   #O_ReadyForOperation := #ReadyForOperation;
END_REGION

REGION Network 49: **** 8 - Outputs **** Alarm AB Condition
   // Alarm AB Condition
   #O_AlarmABCondition := #MovFuncAlmCond OR #StopPosAlmCond OR #MotorLoopAlarmCond OR #LowSpeedSetDetMissingCond OR #LowSpeedResDetMissingCond;
   #AlarmABCondition := #O_AlarmABCondition;
END_REGION

REGION Network 50: **** 9 - Alarm Summary **** Alarm A
   // Alarms A
   #AlarmA := #AA_MotorProtection OR #AA_SafetySwitch OR #AA_NoBusControl;
END_REGION

REGION Network 51: **** 9 - Alarm Summary **** Alarm B
   // Alarms B
   #AlarmB := #AB_TwoDetAlm OR #AB_KeepPosSetAlm OR #AB_KeepPosResAlm OR #AB_OvtSetAlm OR #AB_OvtResAlm OR #AB_LSpeedDetSetMissing OR #AB_LSpeedDetResMissing OR #AB_Alarm OR #AB_STO;
END_REGION

REGION Network 52: **** 9 - Alarm Summary **** Alarm C
   // Alarms C
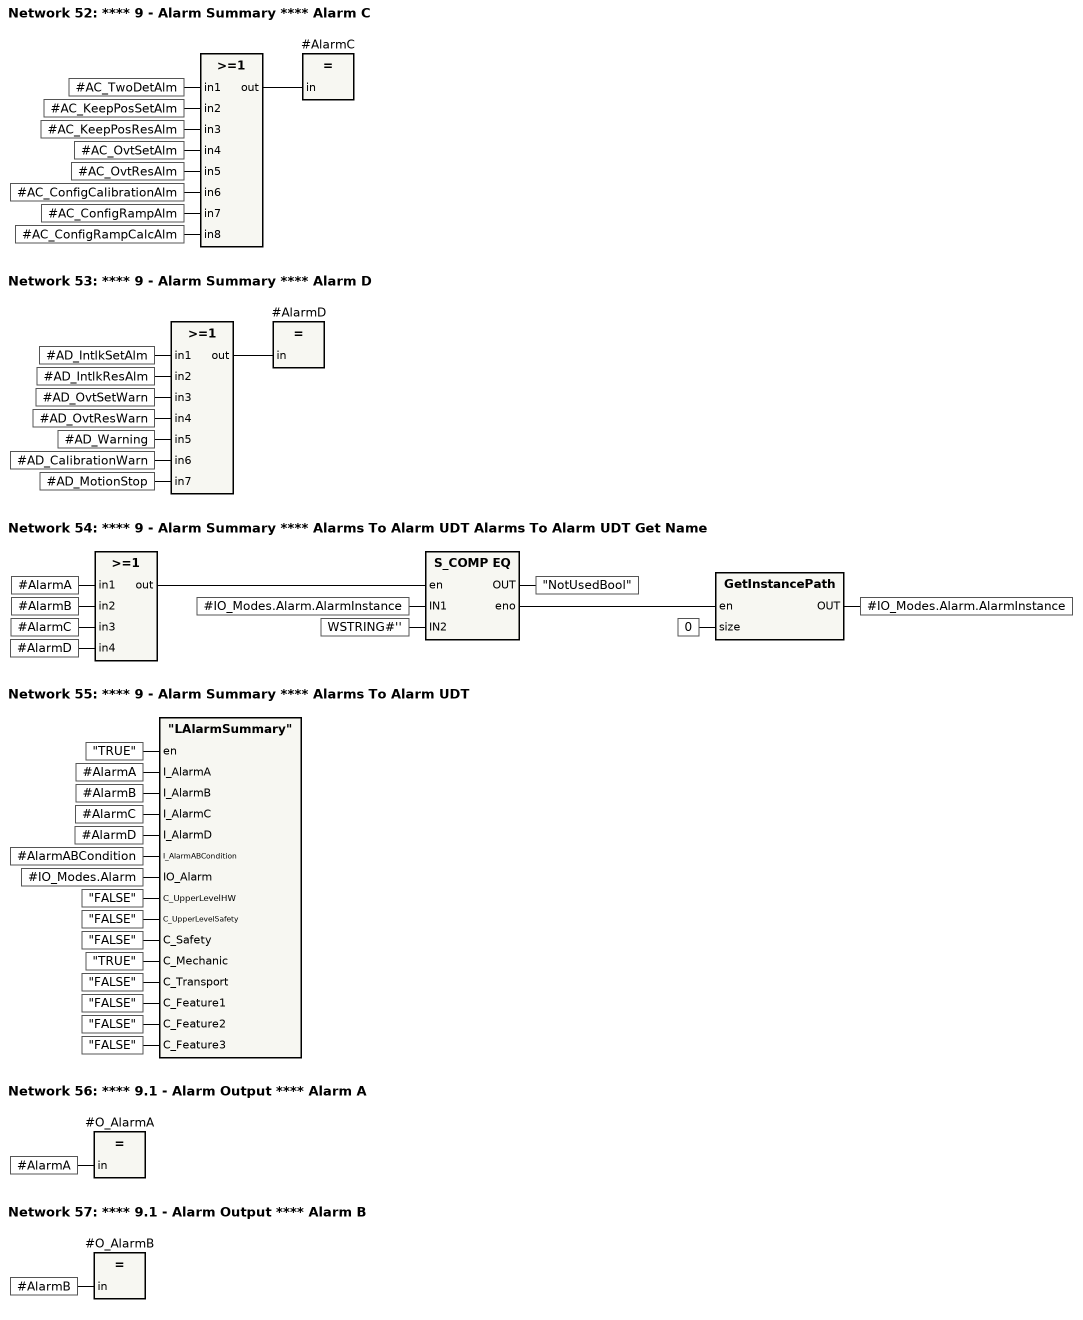
   #AlarmC := #AC_TwoDetAlm OR #AC_KeepPosSetAlm OR #AC_KeepPosResAlm OR #AC_OvtSetAlm OR #AC_OvtResAlm OR #AC_ConfigCalibrationAlm OR #AC_ConfigRampAlm OR #AC_ConfigRampCalcAlm;
END_REGION

REGION Network 53: **** 9 - Alarm Summary **** Alarm D
   // Alarms D
   #AlarmD := #AD_IntlkSetAlm OR #AD_IntlkResAlm OR #AD_OvtSetWarn OR #AD_OvtResWarn OR #AD_Warning OR #AD_CalibrationWarn OR #AD_MotionStop;
END_REGION

REGION Network 54: **** 9 - Alarm Summary **** Alarms To Alarm UDT Alarms To Alarm UDT Get Name
   // Alarm D
   S_COMP(EN := #AlarmA OR #AlarmB OR #AlarmC OR #AlarmD,
          IN1 := #IO_Modes.Alarm.AlarmInstance,
          IN2 := WSTRING#'',
          OUT => "NotUsedBool",
          ENO => #_w1);
   IF #_w1 THEN GetInstancePath(size := 0, OUT => #IO_Modes.Alarm.AlarmInstance); END_IF;
END_REGION

REGION Network 55: **** 9 - Alarm Summary **** Alarms To Alarm UDT
   // Alarm D
   IF "TRUE" THEN
       "LAlarmSummary"(I_AlarmA := #AlarmA,
                       I_AlarmB := #AlarmB,
                       I_AlarmC := #AlarmC,
                       I_AlarmD := #AlarmD,
                       I_AlarmABCondition := #AlarmABCondition,
                       IO_Alarm := #IO_Modes.Alarm,
                       C_UpperLevelHW := "FALSE",
                       C_UpperLevelSafety := "FALSE",
                       C_Safety := "FALSE",
                       C_Mechanic := "TRUE",
                       C_Transport := "FALSE",
                       C_Feature1 := "FALSE",
                       C_Feature2 := "FALSE",
                       C_Feature3 := "FALSE");
   END_IF;
END_REGION

REGION Network 56: **** 9.1 - Alarm Output **** Alarm A
   // Alarm A
   #O_AlarmA := #AlarmA;
END_REGION

REGION Network 57: **** 9.1 - Alarm Output **** Alarm B
   // Alarm B
   #O_AlarmB := #AlarmB;
END_REGION

REGION Network 58: **** 9.1 - Alarm Output **** Alarm C
   // Alarm C
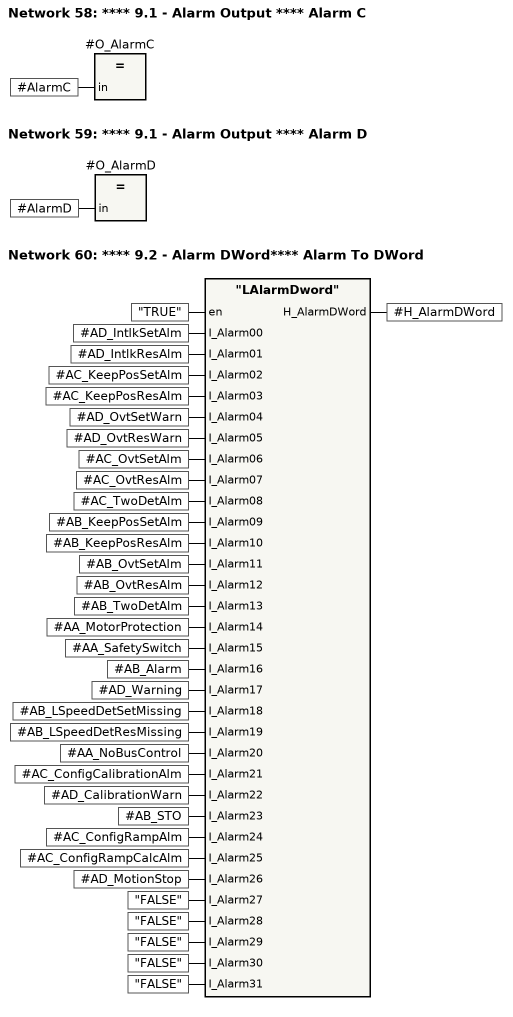
   #O_AlarmC := #AlarmC;
END_REGION

REGION Network 59: **** 9.1 - Alarm Output **** Alarm D
   // Alarm D
   #O_AlarmD := #AlarmD;
END_REGION

REGION Network 60: **** 9.2 - Alarm DWord**** Alarm To DWord
   // Alarm To Word
   IF "TRUE" THEN
       "LAlarmDword"(I_Alarm00 := #AD_IntlkSetAlm,
                     I_Alarm01 := #AD_IntlkResAlm,
                     I_Alarm02 := #AC_KeepPosSetAlm,
                     I_Alarm03 := #AC_KeepPosResAlm,
                     I_Alarm04 := #AD_OvtSetWarn,
                     I_Alarm05 := #AD_OvtResWarn,
                     I_Alarm06 := #AC_OvtSetAlm,
                     I_Alarm07 := #AC_OvtResAlm,
                     I_Alarm08 := #AC_TwoDetAlm,
                     I_Alarm09 := #AB_KeepPosSetAlm,
                     I_Alarm10 := #AB_KeepPosResAlm,
                     I_Alarm11 := #AB_OvtSetAlm,
                     I_Alarm12 := #AB_OvtResAlm,
                     I_Alarm13 := #AB_TwoDetAlm,
                     I_Alarm14 := #AA_MotorProtection,
                     I_Alarm15 := #AA_SafetySwitch,
                     I_Alarm16 := #AB_Alarm,
                     I_Alarm17 := #AD_Warning,
                     I_Alarm18 := #AB_LSpeedDetSetMissing,
                     I_Alarm19 := #AB_LSpeedDetResMissing,
                     I_Alarm20 := #AA_NoBusControl,
                     I_Alarm21 := #AC_ConfigCalibrationAlm,
                     I_Alarm22 := #AD_CalibrationWarn,
                     I_Alarm23 := #AB_STO,
                     I_Alarm24 := #AC_ConfigRampAlm,
                     I_Alarm25 := #AC_ConfigRampCalcAlm,
                     I_Alarm26 := #AD_MotionStop,
                     I_Alarm27 := "FALSE",
                     I_Alarm28 := "FALSE",
                     I_Alarm29 := "FALSE",
                     I_Alarm30 := "FALSE",
                     I_Alarm31 := "FALSE",
                     H_AlarmDWord => #H_AlarmDWord);
   END_IF;
END_REGION
END_FUNCTION_BLOCK
